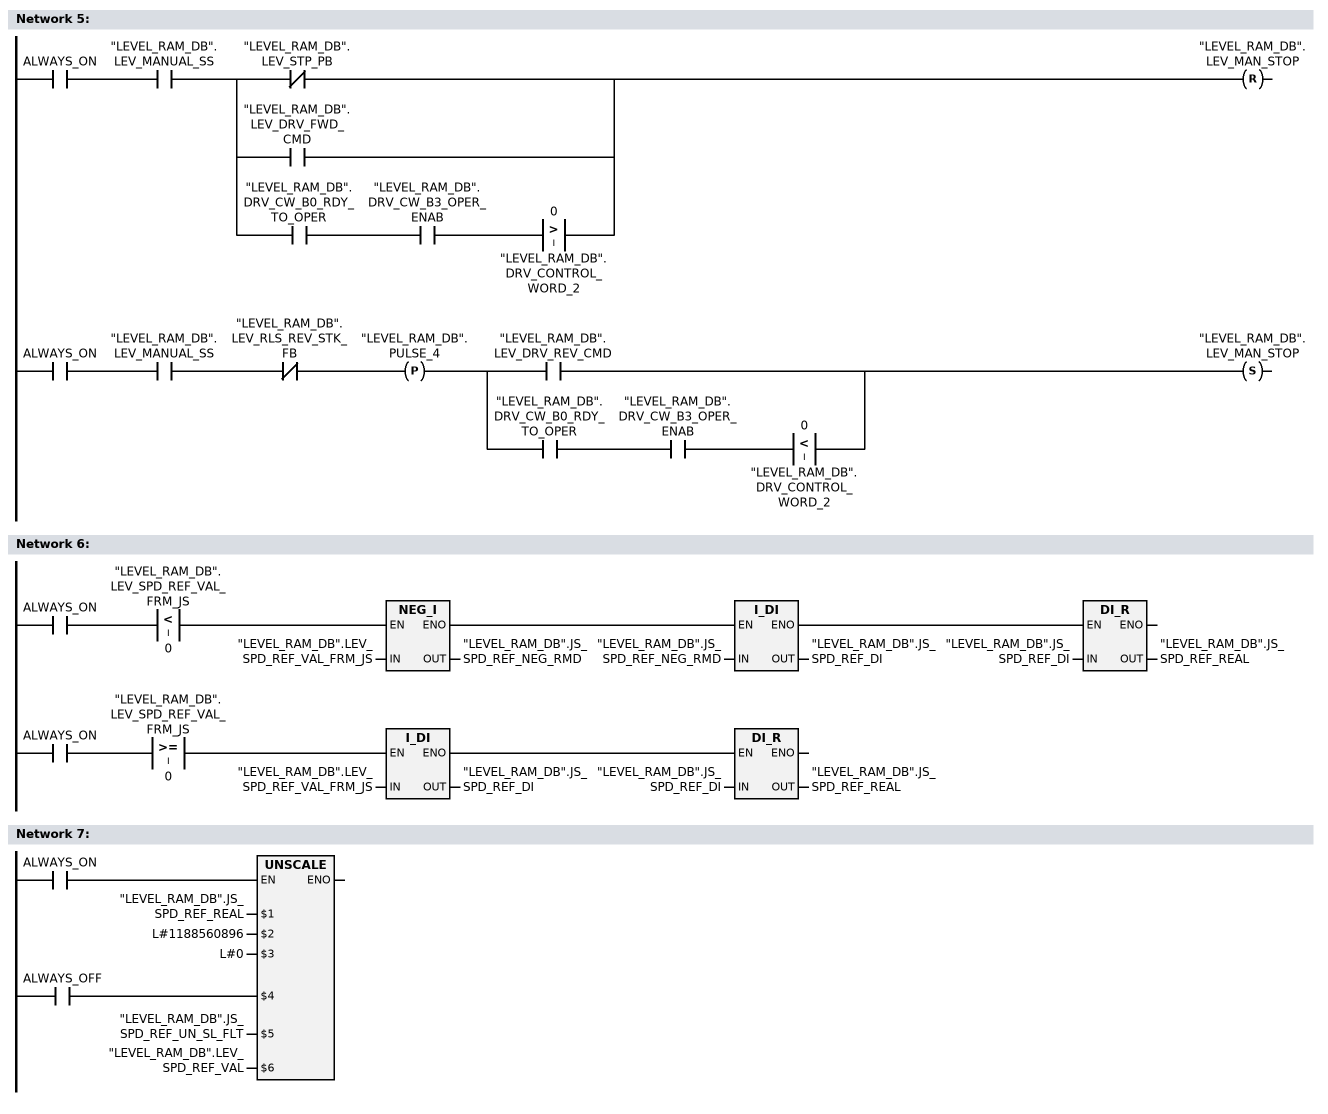
[picture p72: LEVELLER_RAM networks 5-7]
NETWORK
TITLE =
      A     "ALWAYS_ON";
      A     "LEVEL_RAM_DB".LEV_MANUAL_SS;
      =     L 0.0;
      A(;
      A     L 0.0;
      AN    "LEVEL_RAM_DB".LEV_RLS_REV_STK_FB;
      FP    "LEVEL_RAM_DB".PULSE_4;
      );
      A(;
      O     "LEVEL_RAM_DB".LEV_DRV_REV_CMD;
      O;
      A     "LEVEL_RAM_DB".DRV_CW_B0_RDY_TO_OPER;
      A     "LEVEL_RAM_DB".DRV_CW_B3_OPER_ENAB;
      A(;
      L     0;
      L     "LEVEL_RAM_DB".DRV_CONTROL_WORD_2;
      <I;
      );
      );
      S     "LEVEL_RAM_DB".LEV_MAN_STOP;
      A     L 0.0;
      A(;
      ON    "LEVEL_RAM_DB".LEV_STP_PB;
      O     "LEVEL_RAM_DB".LEV_DRV_FWD_CMD;
      O;
      A     "LEVEL_RAM_DB".DRV_CW_B0_RDY_TO_OPER;
      A     "LEVEL_RAM_DB".DRV_CW_B3_OPER_ENAB;
      A(;
      L     0;
      L     "LEVEL_RAM_DB".DRV_CONTROL_WORD_2;
      >I;
      );
      );
      R     "LEVEL_RAM_DB".LEV_MAN_STOP;
NETWORK
TITLE =
      A     "ALWAYS_ON";
      =     L 0.0;
      A(;
      A(;
      A     L 0.0;
      A(;
      L     "LEVEL_RAM_DB".LEV_SPD_REF_VAL_FRM_JS;
      L     0;
      <I;
      );
      JNB   M002;
      L     "LEVEL_RAM_DB".LEV_SPD_REF_VAL_FRM_JS;
      NEGI;
      T     "LEVEL_RAM_DB".JS_SPD_REF_NEG_RMD;
      AN    OV;
      SAVE;
      CLR;
M002: A     BR;
      );
      JNB   M003;
      L     "LEVEL_RAM_DB".JS_SPD_REF_NEG_RMD;
      ITD;
      T     "LEVEL_RAM_DB".JS_SPD_REF_DI;
      SET;
      SAVE;
      CLR;
M003: A     BR;
      );
      JNB   M004;
      L     "LEVEL_RAM_DB".JS_SPD_REF_DI;
      DTR;
      T     "LEVEL_RAM_DB".JS_SPD_REF_REAL;
M004: NOP   0;
      A(;
      A     L 0.0;
      A(;
      L     "LEVEL_RAM_DB".LEV_SPD_REF_VAL_FRM_JS;
      L     0;
      >=I;
      );
      JNB   M005;
      L     "LEVEL_RAM_DB".LEV_SPD_REF_VAL_FRM_JS;
      ITD;
      T     "LEVEL_RAM_DB".JS_SPD_REF_DI;
      SET;
      SAVE;
      CLR;
M005: A     BR;
      );
      JNB   M006;
      L     "LEVEL_RAM_DB".JS_SPD_REF_DI;
      DTR;
      T     "LEVEL_RAM_DB".JS_SPD_REF_REAL;
M006: NOP   0;
NETWORK
TITLE =
      A     "ALWAYS_OFF";
      =     L 0.0;
      BLD   103;
      A     "ALWAYS_ON";
      JNB   M007;
      CALL  "UNSCALE" (
           $1                       := "LEVEL_RAM_DB".JS_SPD_REF_REAL,
           $2                       := L#1188560896,
           $3                       := L#0,
           $4                       := L 0.0,
           $5                       := "LEVEL_RAM_DB".JS_SPD_REF_UN_SL_FLT,
           $6                       := "LEVEL_RAM_DB".LEV_SPD_REF_VAL);
M007: NOP   0;
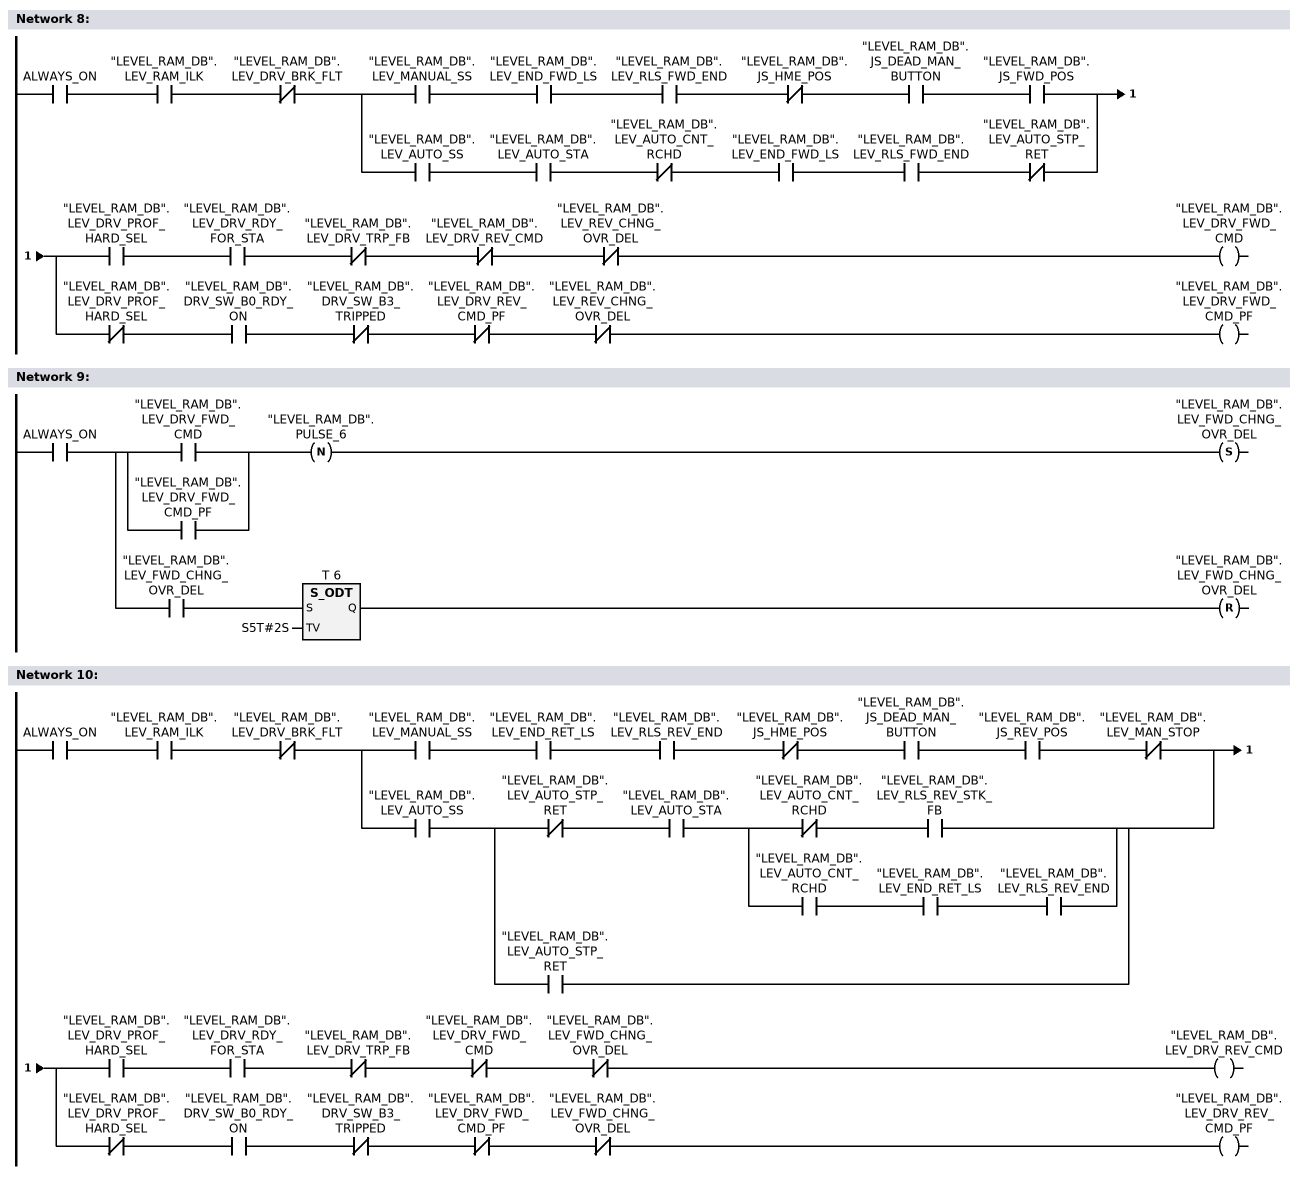
NETWORK
TITLE =
      A     "ALWAYS_ON";
      A     "LEVEL_RAM_DB".LEV_RAM_ILK;
      AN    "LEVEL_RAM_DB".LEV_DRV_BRK_FLT;
      A(;
      A     "LEVEL_RAM_DB".LEV_MANUAL_SS;
      A     "LEVEL_RAM_DB".LEV_END_FWD_LS;
      A     "LEVEL_RAM_DB".LEV_RLS_FWD_END;
      AN    "LEVEL_RAM_DB".JS_HME_POS;
      A     "LEVEL_RAM_DB".JS_DEAD_MAN_BUTTON;
      A     "LEVEL_RAM_DB".JS_FWD_POS;
      O;
      A     "LEVEL_RAM_DB".LEV_AUTO_SS;
      A     "LEVEL_RAM_DB".LEV_AUTO_STA;
      AN    "LEVEL_RAM_DB".LEV_AUTO_CNT_RCHD;
      A     "LEVEL_RAM_DB".LEV_END_FWD_LS;
      A     "LEVEL_RAM_DB".LEV_RLS_FWD_END;
      AN    "LEVEL_RAM_DB".LEV_AUTO_STP_RET;
      );
      =     L 0.0;
      A     L 0.0;
      A     "LEVEL_RAM_DB".LEV_DRV_PROF_HARD_SEL;
      A     "LEVEL_RAM_DB".LEV_DRV_RDY_FOR_STA;
      AN    "LEVEL_RAM_DB".LEV_DRV_TRP_FB;
      AN    "LEVEL_RAM_DB".LEV_DRV_REV_CMD;
      AN    "LEVEL_RAM_DB".LEV_REV_CHNG_OVR_DEL;
      =     "LEVEL_RAM_DB".LEV_DRV_FWD_CMD;
      A     L 0.0;
      AN    "LEVEL_RAM_DB".LEV_DRV_PROF_HARD_SEL;
      A     "LEVEL_RAM_DB".DRV_SW_B0_RDY_ON;
      AN    "LEVEL_RAM_DB".DRV_SW_B3_TRIPPED;
      AN    "LEVEL_RAM_DB".LEV_DRV_REV_CMD_PF;
      AN    "LEVEL_RAM_DB".LEV_REV_CHNG_OVR_DEL;
      =     "LEVEL_RAM_DB".LEV_DRV_FWD_CMD_PF;
NETWORK
TITLE =
      A     "ALWAYS_ON";
      =     L 0.0;
      A     L 0.0;
      A(;
      O     "LEVEL_RAM_DB".LEV_DRV_FWD_CMD;
      O     "LEVEL_RAM_DB".LEV_DRV_FWD_CMD_PF;
      );
      FN    "LEVEL_RAM_DB".PULSE_6;
      S     "LEVEL_RAM_DB".LEV_FWD_CHNG_OVR_DEL;
      A     L 0.0;
      A     "LEVEL_RAM_DB".LEV_FWD_CHNG_OVR_DEL;
      L     S5T#2S;
      SD    T 6;
      NOP   0;
      NOP   0;
      NOP   0;
      A     T 6;
      R     "LEVEL_RAM_DB".LEV_FWD_CHNG_OVR_DEL;
NETWORK
TITLE =
      A     "ALWAYS_ON";
      A     "LEVEL_RAM_DB".LEV_RAM_ILK;
      AN    "LEVEL_RAM_DB".LEV_DRV_BRK_FLT;
      A(;
      A     "LEVEL_RAM_DB".LEV_MANUAL_SS;
      A     "LEVEL_RAM_DB".LEV_END_RET_LS;
      A     "LEVEL_RAM_DB".LEV_RLS_REV_END;
      AN    "LEVEL_RAM_DB".JS_HME_POS;
      A     "LEVEL_RAM_DB".JS_DEAD_MAN_BUTTON;
      A     "LEVEL_RAM_DB".JS_REV_POS;
      AN    "LEVEL_RAM_DB".LEV_MAN_STOP;
      O;
      A     "LEVEL_RAM_DB".LEV_AUTO_SS;
      A(;
      AN    "LEVEL_RAM_DB".LEV_AUTO_STP_RET;
      A     "LEVEL_RAM_DB".LEV_AUTO_STA;
      A(;
      AN    "LEVEL_RAM_DB".LEV_AUTO_CNT_RCHD;
      A     "LEVEL_RAM_DB".LEV_RLS_REV_STK_FB;
      O;
      A     "LEVEL_RAM_DB".LEV_AUTO_CNT_RCHD;
      A     "LEVEL_RAM_DB".LEV_END_RET_LS;
      A     "LEVEL_RAM_DB".LEV_RLS_REV_END;
      );
      O     "LEVEL_RAM_DB".LEV_AUTO_STP_RET;
      );
      );
      =     L 0.0;
      A     L 0.0;
      A     "LEVEL_RAM_DB".LEV_DRV_PROF_HARD_SEL;
      A     "LEVEL_RAM_DB".LEV_DRV_RDY_FOR_STA;
      AN    "LEVEL_RAM_DB".LEV_DRV_TRP_FB;
      AN    "LEVEL_RAM_DB".LEV_DRV_FWD_CMD;
      AN    "LEVEL_RAM_DB".LEV_FWD_CHNG_OVR_DEL;
      =     "LEVEL_RAM_DB".LEV_DRV_REV_CMD;
      A     L 0.0;
      AN    "LEVEL_RAM_DB".LEV_DRV_PROF_HARD_SEL;
      A     "LEVEL_RAM_DB".DRV_SW_B0_RDY_ON;
      AN    "LEVEL_RAM_DB".DRV_SW_B3_TRIPPED;
      AN    "LEVEL_RAM_DB".LEV_DRV_FWD_CMD_PF;
      AN    "LEVEL_RAM_DB".LEV_FWD_CHNG_OVR_DEL;
      =     "LEVEL_RAM_DB".LEV_DRV_REV_CMD_PF;
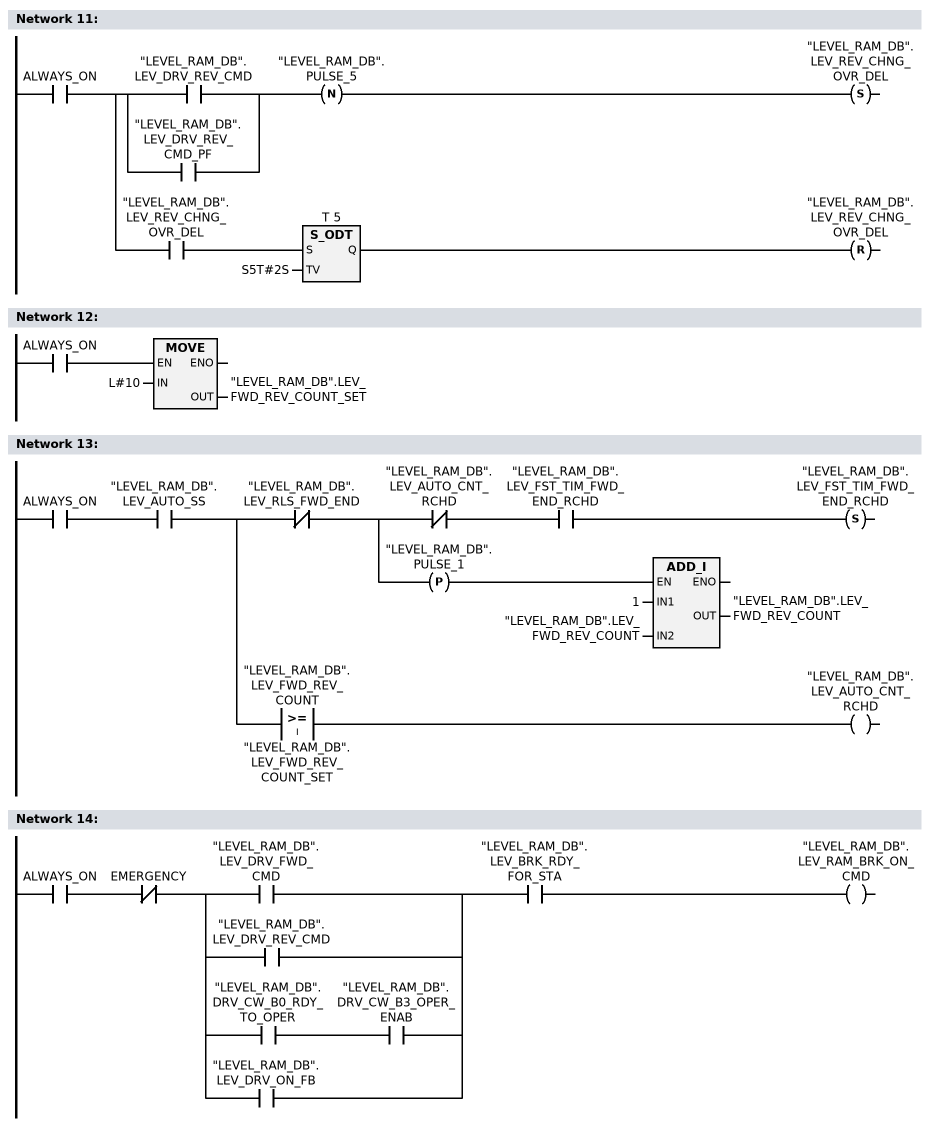
NETWORK
TITLE =
      A     "ALWAYS_ON";
      =     L 0.0;
      A     L 0.0;
      A(;
      O     "LEVEL_RAM_DB".LEV_DRV_REV_CMD;
      O     "LEVEL_RAM_DB".LEV_DRV_REV_CMD_PF;
      );
      FN    "LEVEL_RAM_DB".PULSE_5;
      S     "LEVEL_RAM_DB".LEV_REV_CHNG_OVR_DEL;
      A     L 0.0;
      A     "LEVEL_RAM_DB".LEV_REV_CHNG_OVR_DEL;
      L     S5T#2S;
      SD    T 5;
      NOP   0;
      NOP   0;
      NOP   0;
      A     T 5;
      R     "LEVEL_RAM_DB".LEV_REV_CHNG_OVR_DEL;
NETWORK
TITLE =
      A     "ALWAYS_ON";
      JNB   M008;
      L     L#10;
      T     "LEVEL_RAM_DB".LEV_FWD_REV_COUNT_SET;
M008: NOP   0;
NETWORK
TITLE =
      A     "ALWAYS_ON";
      A     "LEVEL_RAM_DB".LEV_AUTO_SS;
      =     L 0.0;
      A     L 0.0;
      AN    "LEVEL_RAM_DB".LEV_RLS_FWD_END;
      =     L 0.1;
      A     L 0.1;
      AN    "LEVEL_RAM_DB".LEV_AUTO_CNT_RCHD;
      A     "LEVEL_RAM_DB".LEV_FST_TIM_FWD_END_RCHD;
      S     "LEVEL_RAM_DB".LEV_FST_TIM_FWD_END_RCHD;
      A     L 0.1;
      FP    "LEVEL_RAM_DB".PULSE_1;
      JNB   M009;
      L     1;
      L     "LEVEL_RAM_DB".LEV_FWD_REV_COUNT;
      +I;
      T     "LEVEL_RAM_DB".LEV_FWD_REV_COUNT;
M009: NOP   0;
      A     L 0.0;
      A(;
      L     "LEVEL_RAM_DB".LEV_FWD_REV_COUNT;
      L     "LEVEL_RAM_DB".LEV_FWD_REV_COUNT_SET;
      >=I;
      );
      =     "LEVEL_RAM_DB".LEV_AUTO_CNT_RCHD;
NETWORK
TITLE =
      A     "ALWAYS_ON";
      AN    "EMERGENCY";
      A(;
      O     "LEVEL_RAM_DB".LEV_DRV_FWD_CMD;
      O     "LEVEL_RAM_DB".LEV_DRV_REV_CMD;
      O;
      A     "LEVEL_RAM_DB".DRV_CW_B0_RDY_TO_OPER;
      A     "LEVEL_RAM_DB".DRV_CW_B3_OPER_ENAB;
      O     "LEVEL_RAM_DB".LEV_DRV_ON_FB;
      );
      A     "LEVEL_RAM_DB".LEV_BRK_RDY_FOR_STA;
      =     "LEVEL_RAM_DB".LEV_RAM_BRK_ON_CMD;
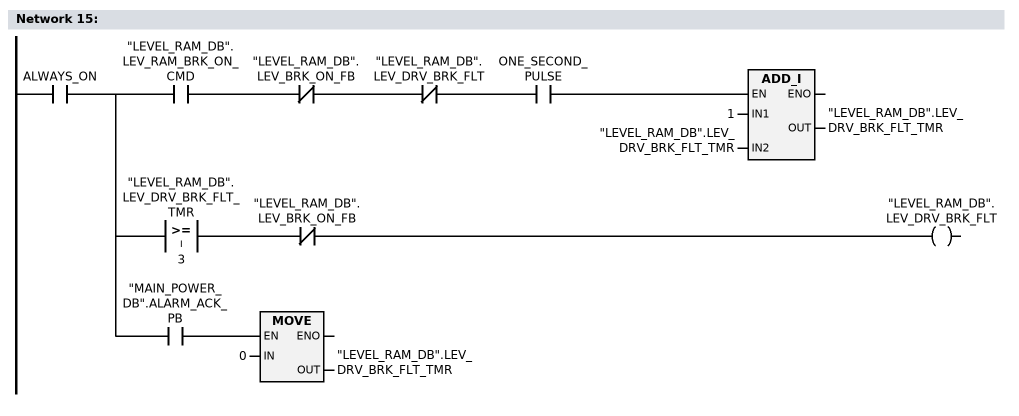
NETWORK
TITLE =
      A     "ALWAYS_ON";
      =     L 0.0;
      A     L 0.0;
      A     "LEVEL_RAM_DB".LEV_RAM_BRK_ON_CMD;
      AN    "LEVEL_RAM_DB".LEV_BRK_ON_FB;
      AN    "LEVEL_RAM_DB".LEV_DRV_BRK_FLT;
      A     "ONE_SECOND_PULSE";
      JNB   M010;
      L     1;
      L     "LEVEL_RAM_DB".LEV_DRV_BRK_FLT_TMR;
      +I;
      T     "LEVEL_RAM_DB".LEV_DRV_BRK_FLT_TMR;
M010: NOP   0;
      A     L 0.0;
      A(;
      L     "LEVEL_RAM_DB".LEV_DRV_BRK_FLT_TMR;
      L     3;
      >=I;
      );
      AN    "LEVEL_RAM_DB".LEV_BRK_ON_FB;
      =     "LEVEL_RAM_DB".LEV_DRV_BRK_FLT;
      A     L 0.0;
      A     "MAIN_POWER_DB".ALARM_ACK_PB;
      JNB   M011;
      L     0;
      T     "LEVEL_RAM_DB".LEV_DRV_BRK_FLT_TMR;
M011: NOP   0;
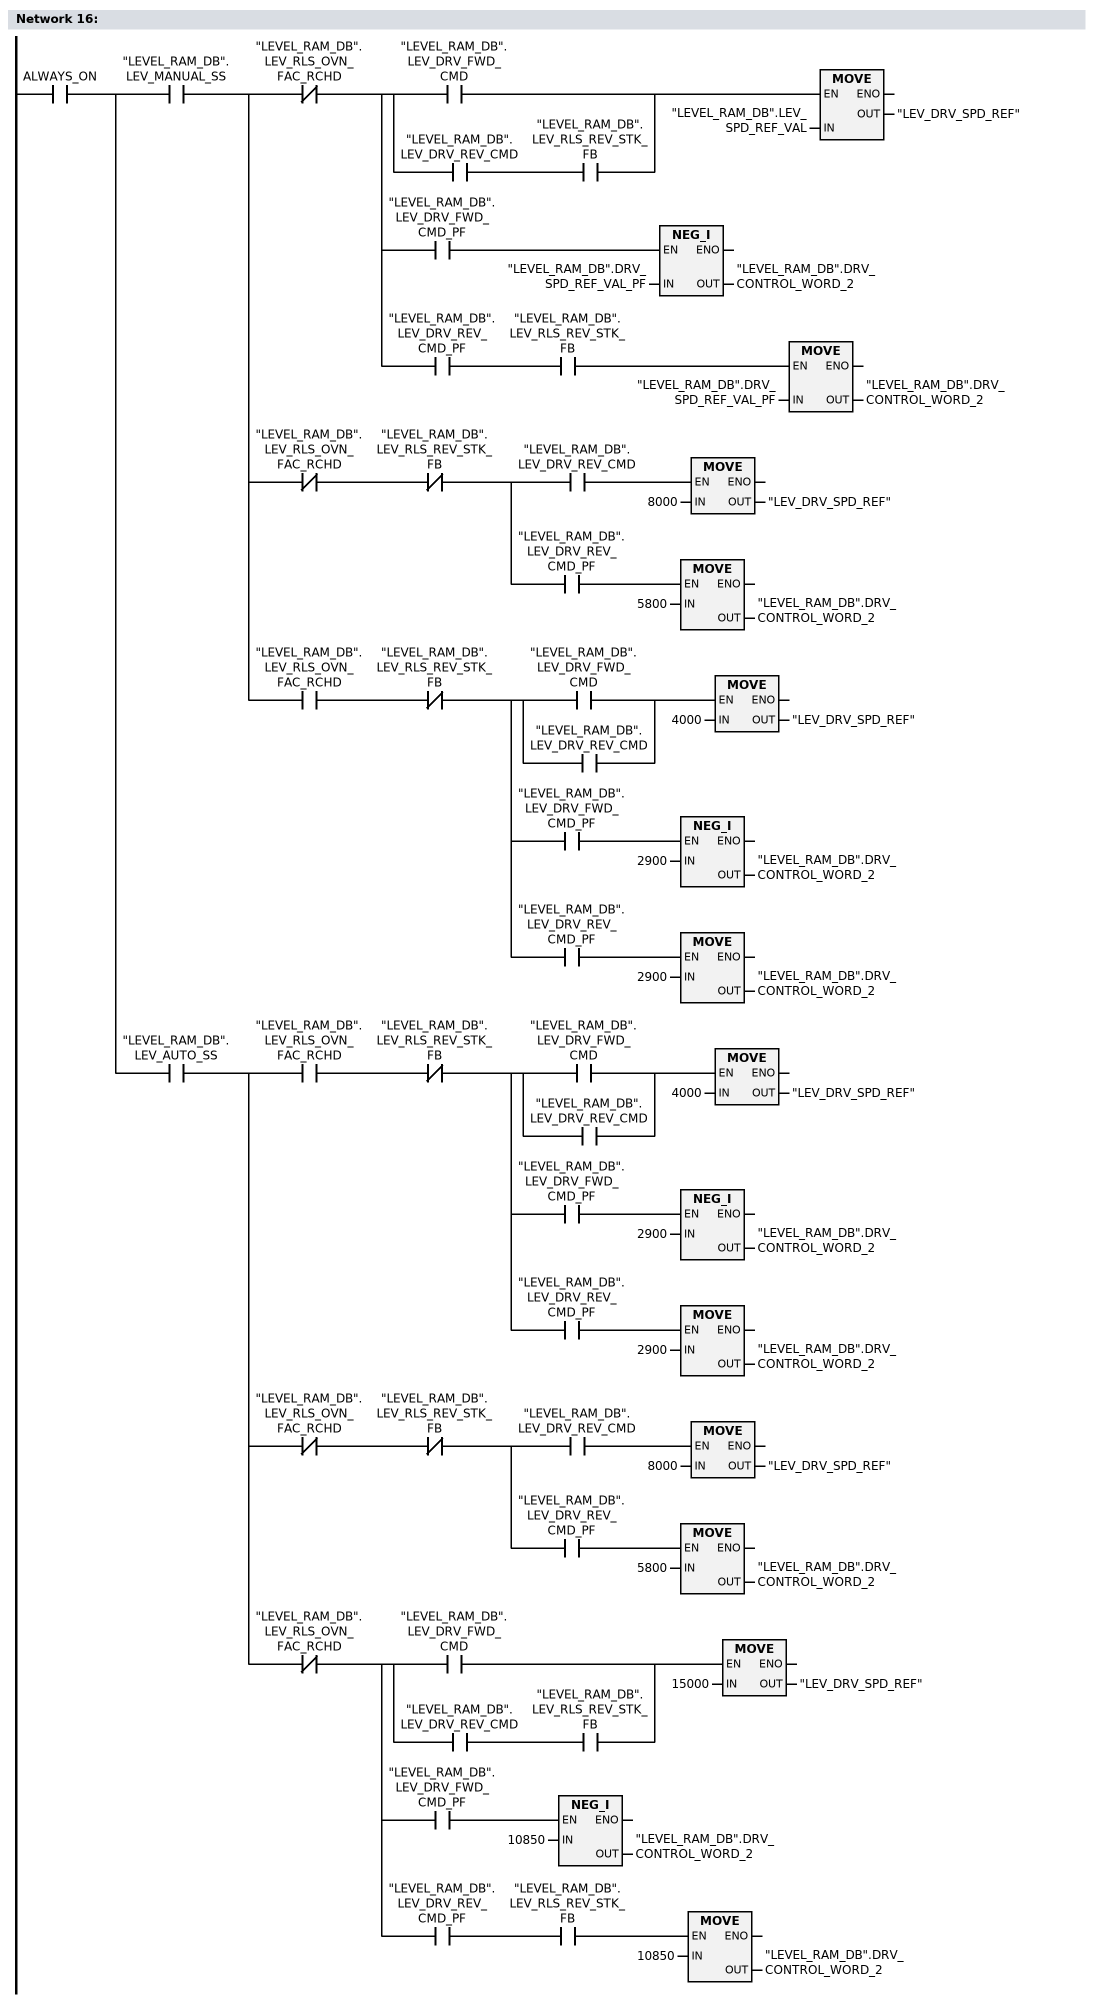
NETWORK
TITLE =
      A     "ALWAYS_ON";
      =     L 0.0;
      A     L 0.0;
      A     "LEVEL_RAM_DB".LEV_MANUAL_SS;
      =     L 0.1;
      A     L 0.1;
      AN    "LEVEL_RAM_DB".LEV_RLS_OVN_FAC_RCHD;
      =     L 0.2;
      A     L 0.2;
      A(;
      O     "LEVEL_RAM_DB".LEV_DRV_FWD_CMD;
      O;
      A     "LEVEL_RAM_DB".LEV_DRV_REV_CMD;
      A     "LEVEL_RAM_DB".LEV_RLS_REV_STK_FB;
      );
      JNB   M012;
      L     "LEVEL_RAM_DB".LEV_SPD_REF_VAL;
      T     "LEV_DRV_SPD_REF";
M012: NOP   0;
      A     L 0.2;
      A     "LEVEL_RAM_DB".LEV_DRV_FWD_CMD_PF;
      JNB   M013;
      L     "LEVEL_RAM_DB".DRV_SPD_REF_VAL_PF;
      NEGI;
      T     "LEVEL_RAM_DB".DRV_CONTROL_WORD_2;
M013: NOP   0;
      A     L 0.2;
      A     "LEVEL_RAM_DB".LEV_DRV_REV_CMD_PF;
      A     "LEVEL_RAM_DB".LEV_RLS_REV_STK_FB;
      JNB   M014;
      L     "LEVEL_RAM_DB".DRV_SPD_REF_VAL_PF;
      T     "LEVEL_RAM_DB".DRV_CONTROL_WORD_2;
M014: NOP   0;
      A     L 0.1;
      AN    "LEVEL_RAM_DB".LEV_RLS_OVN_FAC_RCHD;
      AN    "LEVEL_RAM_DB".LEV_RLS_REV_STK_FB;
      =     L 0.2;
      A     L 0.2;
      A     "LEVEL_RAM_DB".LEV_DRV_REV_CMD;
      JNB   M015;
      L     8000;
      T     "LEV_DRV_SPD_REF";
M015: NOP   0;
      A     L 0.2;
      A     "LEVEL_RAM_DB".LEV_DRV_REV_CMD_PF;
      JNB   M016;
      L     5800;
      T     "LEVEL_RAM_DB".DRV_CONTROL_WORD_2;
M016: NOP   0;
      A     L 0.1;
      A     "LEVEL_RAM_DB".LEV_RLS_OVN_FAC_RCHD;
      AN    "LEVEL_RAM_DB".LEV_RLS_REV_STK_FB;
      =     L 0.2;
      A     L 0.2;
      A(;
      O     "LEVEL_RAM_DB".LEV_DRV_FWD_CMD;
      O     "LEVEL_RAM_DB".LEV_DRV_REV_CMD;
      );
      JNB   M017;
      L     4000;
      T     "LEV_DRV_SPD_REF";
M017: NOP   0;
      A     L 0.2;
      A     "LEVEL_RAM_DB".LEV_DRV_FWD_CMD_PF;
      JNB   M018;
      L     2900;
      NEGI;
      T     "LEVEL_RAM_DB".DRV_CONTROL_WORD_2;
M018: NOP   0;
      A     L 0.2;
      A     "LEVEL_RAM_DB".LEV_DRV_REV_CMD_PF;
      JNB   M019;
      L     2900;
      T     "LEVEL_RAM_DB".DRV_CONTROL_WORD_2;
M019: NOP   0;
      A     L 0.0;
      A     "LEVEL_RAM_DB".LEV_AUTO_SS;
      =     L 0.1;
      A     L 0.1;
      A     "LEVEL_RAM_DB".LEV_RLS_OVN_FAC_RCHD;
      AN    "LEVEL_RAM_DB".LEV_RLS_REV_STK_FB;
      =     L 0.2;
      A     L 0.2;
      A(;
      O     "LEVEL_RAM_DB".LEV_DRV_FWD_CMD;
      O     "LEVEL_RAM_DB".LEV_DRV_REV_CMD;
      );
      JNB   M020;
      L     4000;
      T     "LEV_DRV_SPD_REF";
M020: NOP   0;
      A     L 0.2;
      A     "LEVEL_RAM_DB".LEV_DRV_FWD_CMD_PF;
      JNB   M021;
      L     2900;
      NEGI;
      T     "LEVEL_RAM_DB".DRV_CONTROL_WORD_2;
M021: NOP   0;
      A     L 0.2;
      A     "LEVEL_RAM_DB".LEV_DRV_REV_CMD_PF;
      JNB   M022;
      L     2900;
      T     "LEVEL_RAM_DB".DRV_CONTROL_WORD_2;
M022: NOP   0;
      A     L 0.1;
      AN    "LEVEL_RAM_DB".LEV_RLS_OVN_FAC_RCHD;
      AN    "LEVEL_RAM_DB".LEV_RLS_REV_STK_FB;
      =     L 0.2;
      A     L 0.2;
      A     "LEVEL_RAM_DB".LEV_DRV_REV_CMD;
      JNB   M023;
      L     8000;
      T     "LEV_DRV_SPD_REF";
M023: NOP   0;
      A     L 0.2;
      A     "LEVEL_RAM_DB".LEV_DRV_REV_CMD_PF;
      JNB   M024;
      L     5800;
      T     "LEVEL_RAM_DB".DRV_CONTROL_WORD_2;
M024: NOP   0;
      A     L 0.1;
      AN    "LEVEL_RAM_DB".LEV_RLS_OVN_FAC_RCHD;
      =     L 0.2;
      A     L 0.2;
      A(;
      O     "LEVEL_RAM_DB".LEV_DRV_FWD_CMD;
      O;
      A     "LEVEL_RAM_DB".LEV_DRV_REV_CMD;
      A     "LEVEL_RAM_DB".LEV_RLS_REV_STK_FB;
      );
      JNB   M025;
      L     15000;
      T     "LEV_DRV_SPD_REF";
M025: NOP   0;
      A     L 0.2;
      A     "LEVEL_RAM_DB".LEV_DRV_FWD_CMD_PF;
      JNB   M026;
      L     10850;
      NEGI;
      T     "LEVEL_RAM_DB".DRV_CONTROL_WORD_2;
M026: NOP   0;
      A     L 0.2;
      A     "LEVEL_RAM_DB".LEV_DRV_REV_CMD_PF;
      A     "LEVEL_RAM_DB".LEV_RLS_REV_STK_FB;
      JNB   M027;
      L     10850;
      T     "LEVEL_RAM_DB".DRV_CONTROL_WORD_2;
M027: NOP   0;
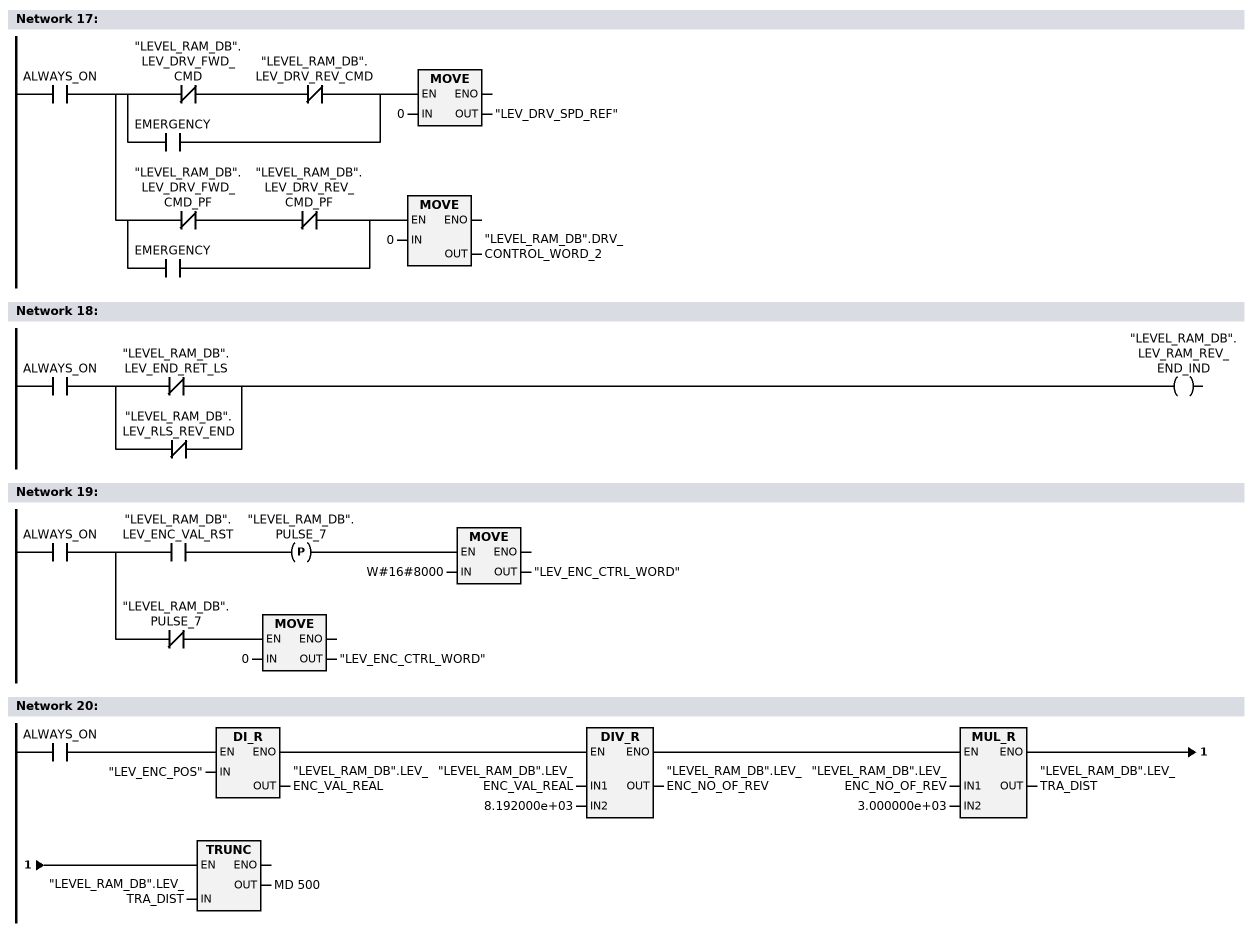
NETWORK
TITLE =
      A     "ALWAYS_ON";
      =     L 0.0;
      A     L 0.0;
      A(;
      AN    "LEVEL_RAM_DB".LEV_DRV_FWD_CMD;
      AN    "LEVEL_RAM_DB".LEV_DRV_REV_CMD;
      O     "EMERGENCY";
      );
      JNB   M028;
      L     0;
      T     "LEV_DRV_SPD_REF";
M028: NOP   0;
      A     L 0.0;
      A(;
      AN    "LEVEL_RAM_DB".LEV_DRV_FWD_CMD_PF;
      AN    "LEVEL_RAM_DB".LEV_DRV_REV_CMD_PF;
      O     "EMERGENCY";
      );
      JNB   M029;
      L     0;
      T     "LEVEL_RAM_DB".DRV_CONTROL_WORD_2;
M029: NOP   0;
NETWORK
TITLE =
      A     "ALWAYS_ON";
      A(;
      ON    "LEVEL_RAM_DB".LEV_END_RET_LS;
      ON    "LEVEL_RAM_DB".LEV_RLS_REV_END;
      );
      =     "LEVEL_RAM_DB".LEV_RAM_REV_END_IND;
NETWORK
TITLE =
      A     "ALWAYS_ON";
      =     L 0.0;
      A     L 0.0;
      A     "LEVEL_RAM_DB".LEV_ENC_VAL_RST;
      FP    "LEVEL_RAM_DB".PULSE_7;
      JNB   M030;
      L     W#16#8000;
      T     "LEV_ENC_CTRL_WORD";
M030: NOP   0;
      A     L 0.0;
      AN    "LEVEL_RAM_DB".PULSE_7;
      JNB   M031;
      L     0;
      T     "LEV_ENC_CTRL_WORD";
M031: NOP   0;
NETWORK
TITLE =
      A(;
      A(;
      A(;
      A     "ALWAYS_ON";
      JNB   M032;
      L     "LEV_ENC_POS";
      DTR;
      T     "LEVEL_RAM_DB".LEV_ENC_VAL_REAL;
      SET;
      SAVE;
      CLR;
M032: A     BR;
      );
      JNB   M033;
      L     "LEVEL_RAM_DB".LEV_ENC_VAL_REAL;
      L     8.192000e+03;
      /R;
      T     "LEVEL_RAM_DB".LEV_ENC_NO_OF_REV;
      AN    OV;
      SAVE;
      CLR;
M033: A     BR;
      );
      JNB   M034;
      L     "LEVEL_RAM_DB".LEV_ENC_NO_OF_REV;
      L     3.000000e+03;
      *R;
      T     "LEVEL_RAM_DB".LEV_TRA_DIST;
      AN    OV;
      SAVE;
      CLR;
M034: A     BR;
      );
      JNB   M035;
      L     "LEVEL_RAM_DB".LEV_TRA_DIST;
      TRUNC;
      T     MD 500;
M035: NOP   0;
END_FUNCTION

FUNCTION "LEVELER_DOOR" : VOID	// FC 6
AUTHOR : Kamillas
VERSION : 0.1
BEGIN
// (block stored without names or comments; labels and parameter names are numbered)
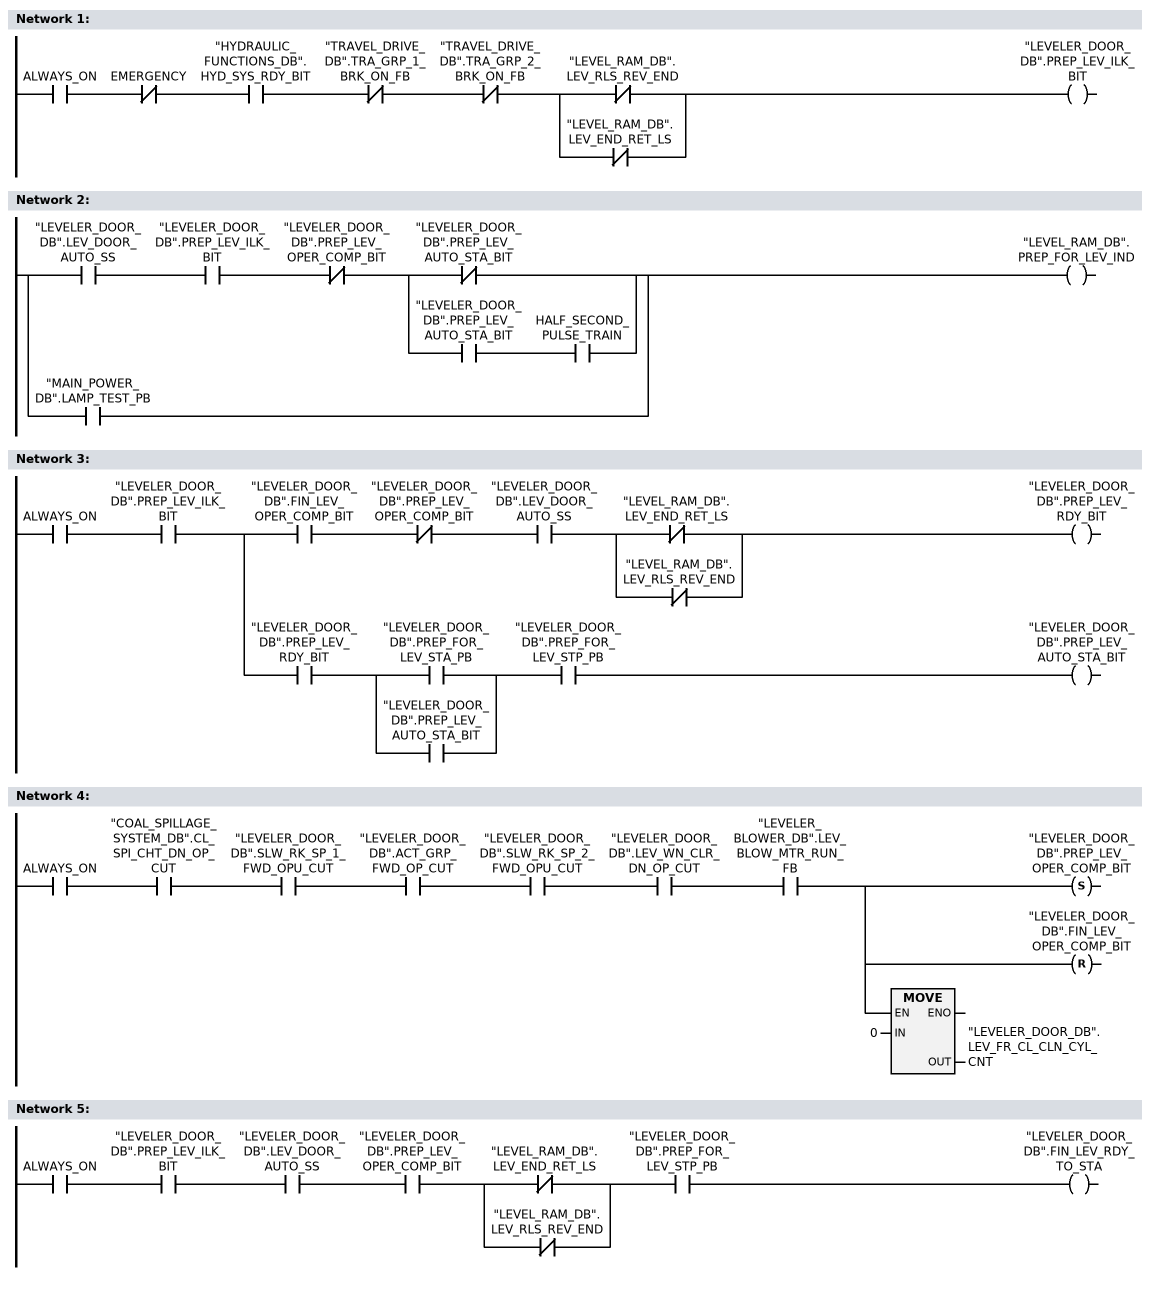
NETWORK
TITLE =
      A     "ALWAYS_ON";
      AN    "EMERGENCY";
      A     "HYDRAULIC_FUNCTIONS_DB".HYD_SYS_RDY_BIT;
      AN    "TRAVEL_DRIVE_DB".TRA_GRP_1_BRK_ON_FB;
      AN    "TRAVEL_DRIVE_DB".TRA_GRP_2_BRK_ON_FB;
      A(;
      ON    "LEVEL_RAM_DB".LEV_RLS_REV_END;
      ON    "LEVEL_RAM_DB".LEV_END_RET_LS;
      );
      =     "LEVELER_DOOR_DB".PREP_LEV_ILK_BIT;
NETWORK
TITLE =
      A     "LEVELER_DOOR_DB".LEV_DOOR_AUTO_SS;
      A     "LEVELER_DOOR_DB".PREP_LEV_ILK_BIT;
      AN    "LEVELER_DOOR_DB".PREP_LEV_OPER_COMP_BIT;
      A(;
      ON    "LEVELER_DOOR_DB".PREP_LEV_AUTO_STA_BIT;
      O;
      A     "LEVELER_DOOR_DB".PREP_LEV_AUTO_STA_BIT;
      A     "HALF_SECOND_PULSE_TRAIN";
      );
      O     "MAIN_POWER_DB".LAMP_TEST_PB;
      =     "LEVEL_RAM_DB".PREP_FOR_LEV_IND;
NETWORK
TITLE =
      A     "ALWAYS_ON";
      A     "LEVELER_DOOR_DB".PREP_LEV_ILK_BIT;
      =     L 0.0;
      A     L 0.0;
      A     "LEVELER_DOOR_DB".FIN_LEV_OPER_COMP_BIT;
      AN    "LEVELER_DOOR_DB".PREP_LEV_OPER_COMP_BIT;
      A     "LEVELER_DOOR_DB".LEV_DOOR_AUTO_SS;
      A(;
      ON    "LEVEL_RAM_DB".LEV_END_RET_LS;
      ON    "LEVEL_RAM_DB".LEV_RLS_REV_END;
      );
      =     "LEVELER_DOOR_DB".PREP_LEV_RDY_BIT;
      A     L 0.0;
      A     "LEVELER_DOOR_DB".PREP_LEV_RDY_BIT;
      A(;
      O     "LEVELER_DOOR_DB".PREP_FOR_LEV_STA_PB;
      O     "LEVELER_DOOR_DB".PREP_LEV_AUTO_STA_BIT;
      );
      A     "LEVELER_DOOR_DB".PREP_FOR_LEV_STP_PB;
      =     "LEVELER_DOOR_DB".PREP_LEV_AUTO_STA_BIT;
NETWORK
TITLE =
      A     "ALWAYS_ON";
      A     "COAL_SPILLAGE_SYSTEM_DB".CL_SPI_CHT_DN_OP_CUT;
      A     "LEVELER_DOOR_DB".SLW_RK_SP_1_FWD_OPU_CUT;
      A     "LEVELER_DOOR_DB".ACT_GRP_FWD_OP_CUT;
      A     "LEVELER_DOOR_DB".SLW_RK_SP_2_FWD_OPU_CUT;
      A     "LEVELER_DOOR_DB".LEV_WN_CLR_DN_OP_CUT;
      A     "LEVELER_BLOWER_DB".LEV_BLOW_MTR_RUN_FB;
      =     L 0.0;
      A     L 0.0;
      BLD   102;
      S     "LEVELER_DOOR_DB".PREP_LEV_OPER_COMP_BIT;
      A     L 0.0;
      BLD   102;
      R     "LEVELER_DOOR_DB".FIN_LEV_OPER_COMP_BIT;
      A     L 0.0;
      JNB   M001;
      L     0;
      T     "LEVELER_DOOR_DB".LEV_FR_CL_CLN_CYL_CNT;
M001: NOP   0;
NETWORK
TITLE =
      A     "ALWAYS_ON";
      A     "LEVELER_DOOR_DB".PREP_LEV_ILK_BIT;
      A     "LEVELER_DOOR_DB".LEV_DOOR_AUTO_SS;
      A     "LEVELER_DOOR_DB".PREP_LEV_OPER_COMP_BIT;
      A(;
      ON    "LEVEL_RAM_DB".LEV_END_RET_LS;
      ON    "LEVEL_RAM_DB".LEV_RLS_REV_END;
      );
      A     "LEVELER_DOOR_DB".PREP_FOR_LEV_STP_PB;
      =     "LEVELER_DOOR_DB".FIN_LEV_RDY_TO_STA;
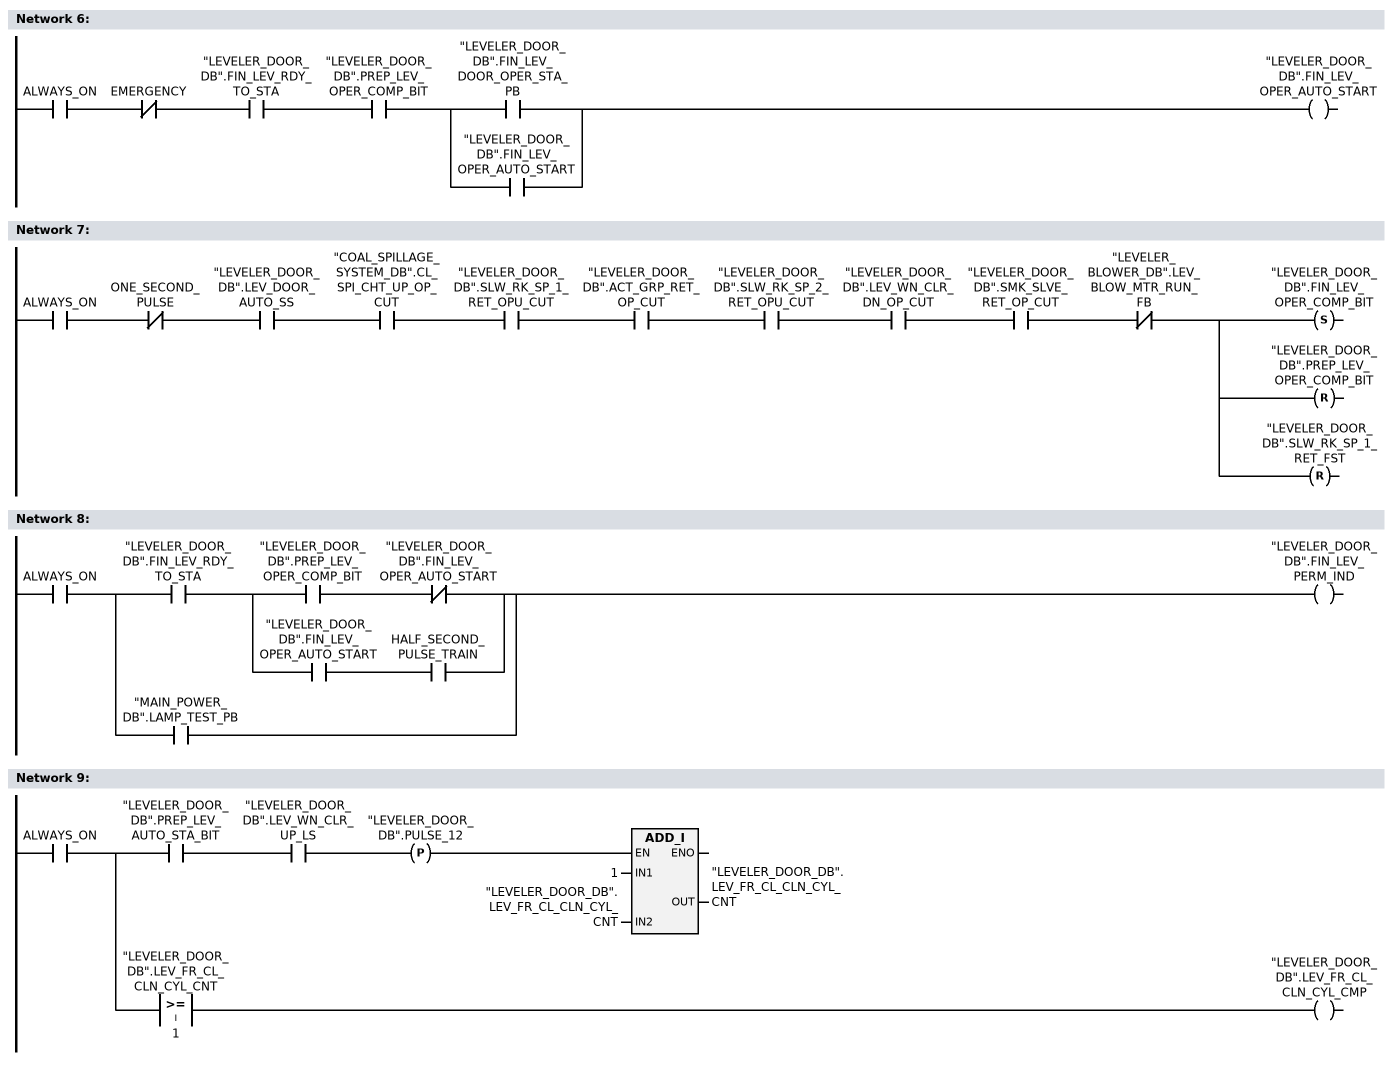
NETWORK
TITLE =
      A     "ALWAYS_ON";
      AN    "EMERGENCY";
      A     "LEVELER_DOOR_DB".FIN_LEV_RDY_TO_STA;
      A     "LEVELER_DOOR_DB".PREP_LEV_OPER_COMP_BIT;
      A(;
      O     "LEVELER_DOOR_DB".FIN_LEV_DOOR_OPER_STA_PB;
      O     "LEVELER_DOOR_DB".FIN_LEV_OPER_AUTO_START;
      );
      =     "LEVELER_DOOR_DB".FIN_LEV_OPER_AUTO_START;
NETWORK
TITLE =
      A     "ALWAYS_ON";
      AN    "ONE_SECOND_PULSE";
      A     "LEVELER_DOOR_DB".LEV_DOOR_AUTO_SS;
      A     "COAL_SPILLAGE_SYSTEM_DB".CL_SPI_CHT_UP_OP_CUT;
      A     "LEVELER_DOOR_DB".SLW_RK_SP_1_RET_OPU_CUT;
      A     "LEVELER_DOOR_DB".ACT_GRP_RET_OP_CUT;
      A     "LEVELER_DOOR_DB".SLW_RK_SP_2_RET_OPU_CUT;
      A     "LEVELER_DOOR_DB".LEV_WN_CLR_DN_OP_CUT;
      A     "LEVELER_DOOR_DB".SMK_SLVE_RET_OP_CUT;
      AN    "LEVELER_BLOWER_DB".LEV_BLOW_MTR_RUN_FB;
      S     "LEVELER_DOOR_DB".FIN_LEV_OPER_COMP_BIT;
      R     "LEVELER_DOOR_DB".PREP_LEV_OPER_COMP_BIT;
      R     "LEVELER_DOOR_DB".SLW_RK_SP_1_RET_FST;
NETWORK
TITLE =
      A     "ALWAYS_ON";
      A(;
      A     "LEVELER_DOOR_DB".FIN_LEV_RDY_TO_STA;
      A(;
      A     "LEVELER_DOOR_DB".PREP_LEV_OPER_COMP_BIT;
      AN    "LEVELER_DOOR_DB".FIN_LEV_OPER_AUTO_START;
      O;
      A     "LEVELER_DOOR_DB".FIN_LEV_OPER_AUTO_START;
      A     "HALF_SECOND_PULSE_TRAIN";
      );
      O     "MAIN_POWER_DB".LAMP_TEST_PB;
      );
      =     "LEVELER_DOOR_DB".FIN_LEV_PERM_IND;
NETWORK
TITLE =
      A     "ALWAYS_ON";
      =     L 0.0;
      A     L 0.0;
      A     "LEVELER_DOOR_DB".PREP_LEV_AUTO_STA_BIT;
      A     "LEVELER_DOOR_DB".LEV_WN_CLR_UP_LS;
      FP    "LEVELER_DOOR_DB".PULSE_12;
      JNB   M002;
      L     1;
      L     "LEVELER_DOOR_DB".LEV_FR_CL_CLN_CYL_CNT;
      +I;
      T     "LEVELER_DOOR_DB".LEV_FR_CL_CLN_CYL_CNT;
M002: NOP   0;
      A     L 0.0;
      A(;
      L     "LEVELER_DOOR_DB".LEV_FR_CL_CLN_CYL_CNT;
      L     1;
      >=I;
      );
      =     "LEVELER_DOOR_DB".LEV_FR_CL_CLN_CYL_CMP;
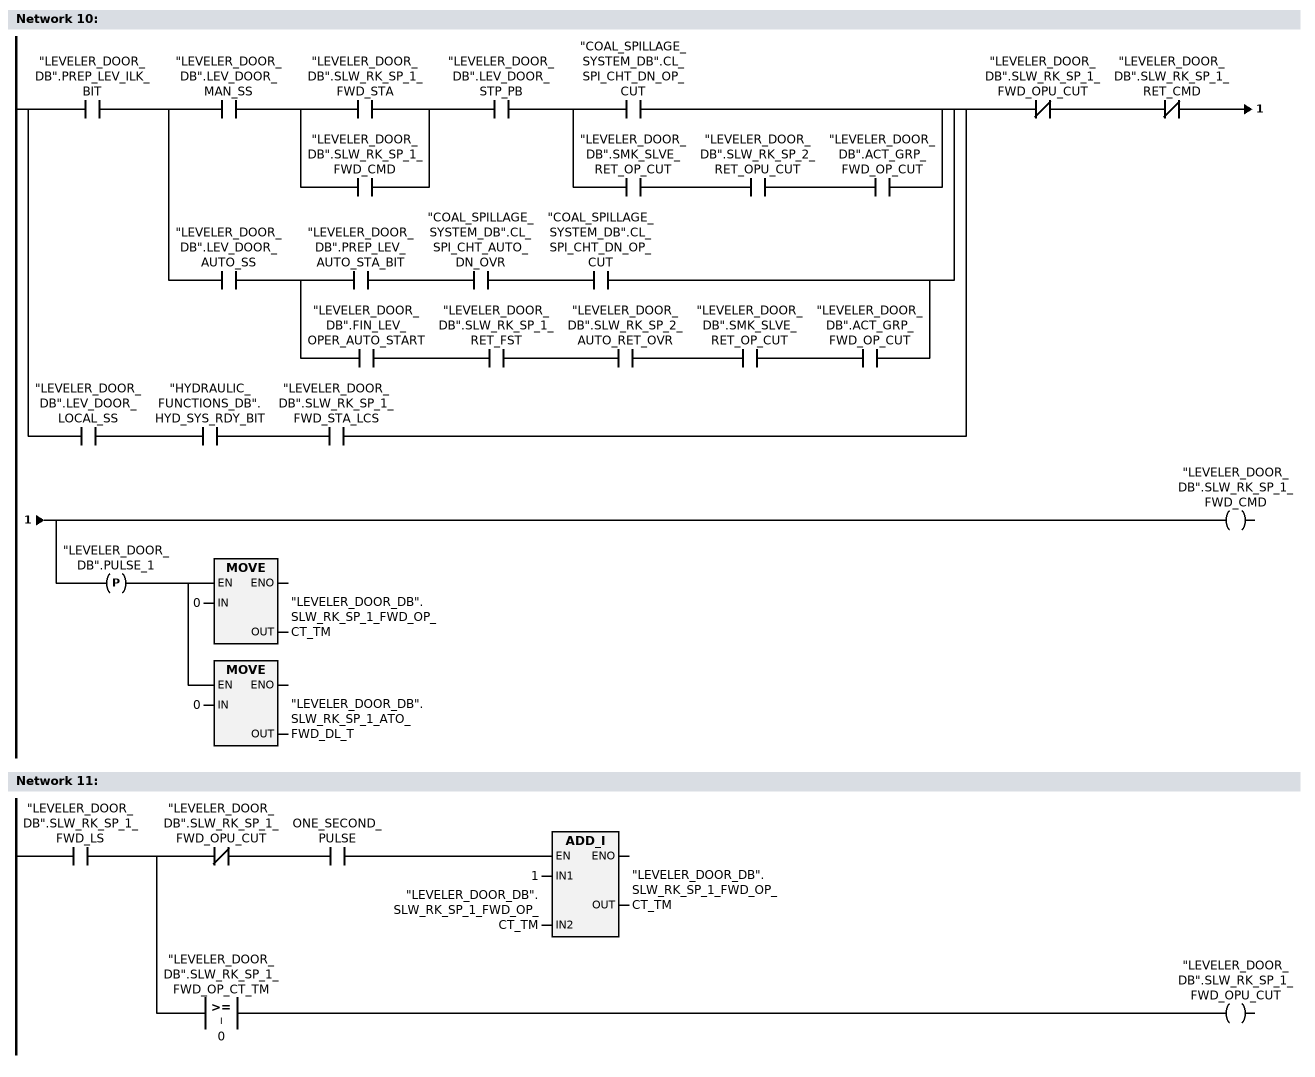
NETWORK
TITLE =
      A(;
      A     "LEVELER_DOOR_DB".PREP_LEV_ILK_BIT;
      A(;
      A     "LEVELER_DOOR_DB".LEV_DOOR_MAN_SS;
      A(;
      O     "LEVELER_DOOR_DB".SLW_RK_SP_1_FWD_STA;
      O     "LEVELER_DOOR_DB".SLW_RK_SP_1_FWD_CMD;
      );
      A     "LEVELER_DOOR_DB".LEV_DOOR_STP_PB;
      A(;
      O     "COAL_SPILLAGE_SYSTEM_DB".CL_SPI_CHT_DN_OP_CUT;
      O;
      A     "LEVELER_DOOR_DB".SMK_SLVE_RET_OP_CUT;
      A     "LEVELER_DOOR_DB".SLW_RK_SP_2_RET_OPU_CUT;
      A     "LEVELER_DOOR_DB".ACT_GRP_FWD_OP_CUT;
      );
      O;
      A     "LEVELER_DOOR_DB".LEV_DOOR_AUTO_SS;
      A(;
      A     "LEVELER_DOOR_DB".PREP_LEV_AUTO_STA_BIT;
      A     "COAL_SPILLAGE_SYSTEM_DB".CL_SPI_CHT_AUTO_DN_OVR;
      A     "COAL_SPILLAGE_SYSTEM_DB".CL_SPI_CHT_DN_OP_CUT;
      O;
      A     "LEVELER_DOOR_DB".FIN_LEV_OPER_AUTO_START;
      A     "LEVELER_DOOR_DB".SLW_RK_SP_1_RET_FST;
      A     "LEVELER_DOOR_DB".SLW_RK_SP_2_AUTO_RET_OVR;
      A     "LEVELER_DOOR_DB".SMK_SLVE_RET_OP_CUT;
      A     "LEVELER_DOOR_DB".ACT_GRP_FWD_OP_CUT;
      );
      );
      O;
      A     "LEVELER_DOOR_DB".LEV_DOOR_LOCAL_SS;
      A     "HYDRAULIC_FUNCTIONS_DB".HYD_SYS_RDY_BIT;
      A     "LEVELER_DOOR_DB".SLW_RK_SP_1_FWD_STA_LCS;
      );
      AN    "LEVELER_DOOR_DB".SLW_RK_SP_1_FWD_OPU_CUT;
      AN    "LEVELER_DOOR_DB".SLW_RK_SP_1_RET_CMD;
      =     L 0.0;
      A     L 0.0;
      BLD   102;
      =     "LEVELER_DOOR_DB".SLW_RK_SP_1_FWD_CMD;
      A     L 0.0;
      FP    "LEVELER_DOOR_DB".PULSE_1;
      =     L 0.1;
      A     L 0.1;
      JNB   M003;
      L     0;
      T     "LEVELER_DOOR_DB".SLW_RK_SP_1_FWD_OP_CT_TM;
M003: NOP   0;
      A     L 0.1;
      JNB   M004;
      L     0;
      T     "LEVELER_DOOR_DB".SLW_RK_SP_1_ATO_FWD_DL_T;
M004: NOP   0;
NETWORK
TITLE =
      A     "LEVELER_DOOR_DB".SLW_RK_SP_1_FWD_LS;
      =     L 0.0;
      A     L 0.0;
      AN    "LEVELER_DOOR_DB".SLW_RK_SP_1_FWD_OPU_CUT;
      A     "ONE_SECOND_PULSE";
      JNB   M005;
      L     1;
      L     "LEVELER_DOOR_DB".SLW_RK_SP_1_FWD_OP_CT_TM;
      +I;
      T     "LEVELER_DOOR_DB".SLW_RK_SP_1_FWD_OP_CT_TM;
M005: NOP   0;
      A     L 0.0;
      A(;
      L     "LEVELER_DOOR_DB".SLW_RK_SP_1_FWD_OP_CT_TM;
      L     0;
      >=I;
      );
      =     "LEVELER_DOOR_DB".SLW_RK_SP_1_FWD_OPU_CUT;
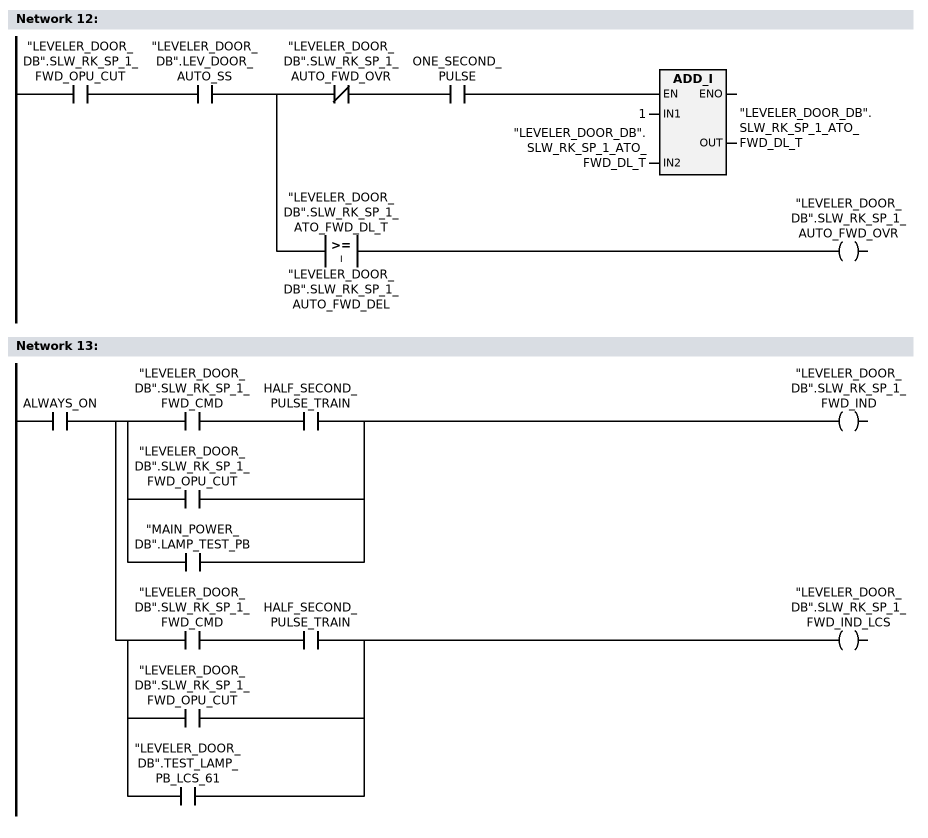
NETWORK
TITLE =
      A     "LEVELER_DOOR_DB".SLW_RK_SP_1_FWD_OPU_CUT;
      A     "LEVELER_DOOR_DB".LEV_DOOR_AUTO_SS;
      =     L 0.0;
      A     L 0.0;
      AN    "LEVELER_DOOR_DB".SLW_RK_SP_1_AUTO_FWD_OVR;
      A     "ONE_SECOND_PULSE";
      JNB   M006;
      L     1;
      L     "LEVELER_DOOR_DB".SLW_RK_SP_1_ATO_FWD_DL_T;
      +I;
      T     "LEVELER_DOOR_DB".SLW_RK_SP_1_ATO_FWD_DL_T;
M006: NOP   0;
      A     L 0.0;
      A(;
      L     "LEVELER_DOOR_DB".SLW_RK_SP_1_ATO_FWD_DL_T;
      L     "LEVELER_DOOR_DB".SLW_RK_SP_1_AUTO_FWD_DEL;
      >=I;
      );
      =     "LEVELER_DOOR_DB".SLW_RK_SP_1_AUTO_FWD_OVR;
NETWORK
TITLE =
      A     "ALWAYS_ON";
      =     L 0.0;
      A     L 0.0;
      A(;
      A     "LEVELER_DOOR_DB".SLW_RK_SP_1_FWD_CMD;
      A     "HALF_SECOND_PULSE_TRAIN";
      O     "LEVELER_DOOR_DB".SLW_RK_SP_1_FWD_OPU_CUT;
      O     "MAIN_POWER_DB".LAMP_TEST_PB;
      );
      =     "LEVELER_DOOR_DB".SLW_RK_SP_1_FWD_IND;
      A     L 0.0;
      A(;
      A     "LEVELER_DOOR_DB".SLW_RK_SP_1_FWD_CMD;
      A     "HALF_SECOND_PULSE_TRAIN";
      O     "LEVELER_DOOR_DB".SLW_RK_SP_1_FWD_OPU_CUT;
      O     "LEVELER_DOOR_DB".TEST_LAMP_PB_LCS_61;
      );
      =     "LEVELER_DOOR_DB".SLW_RK_SP_1_FWD_IND_LCS;
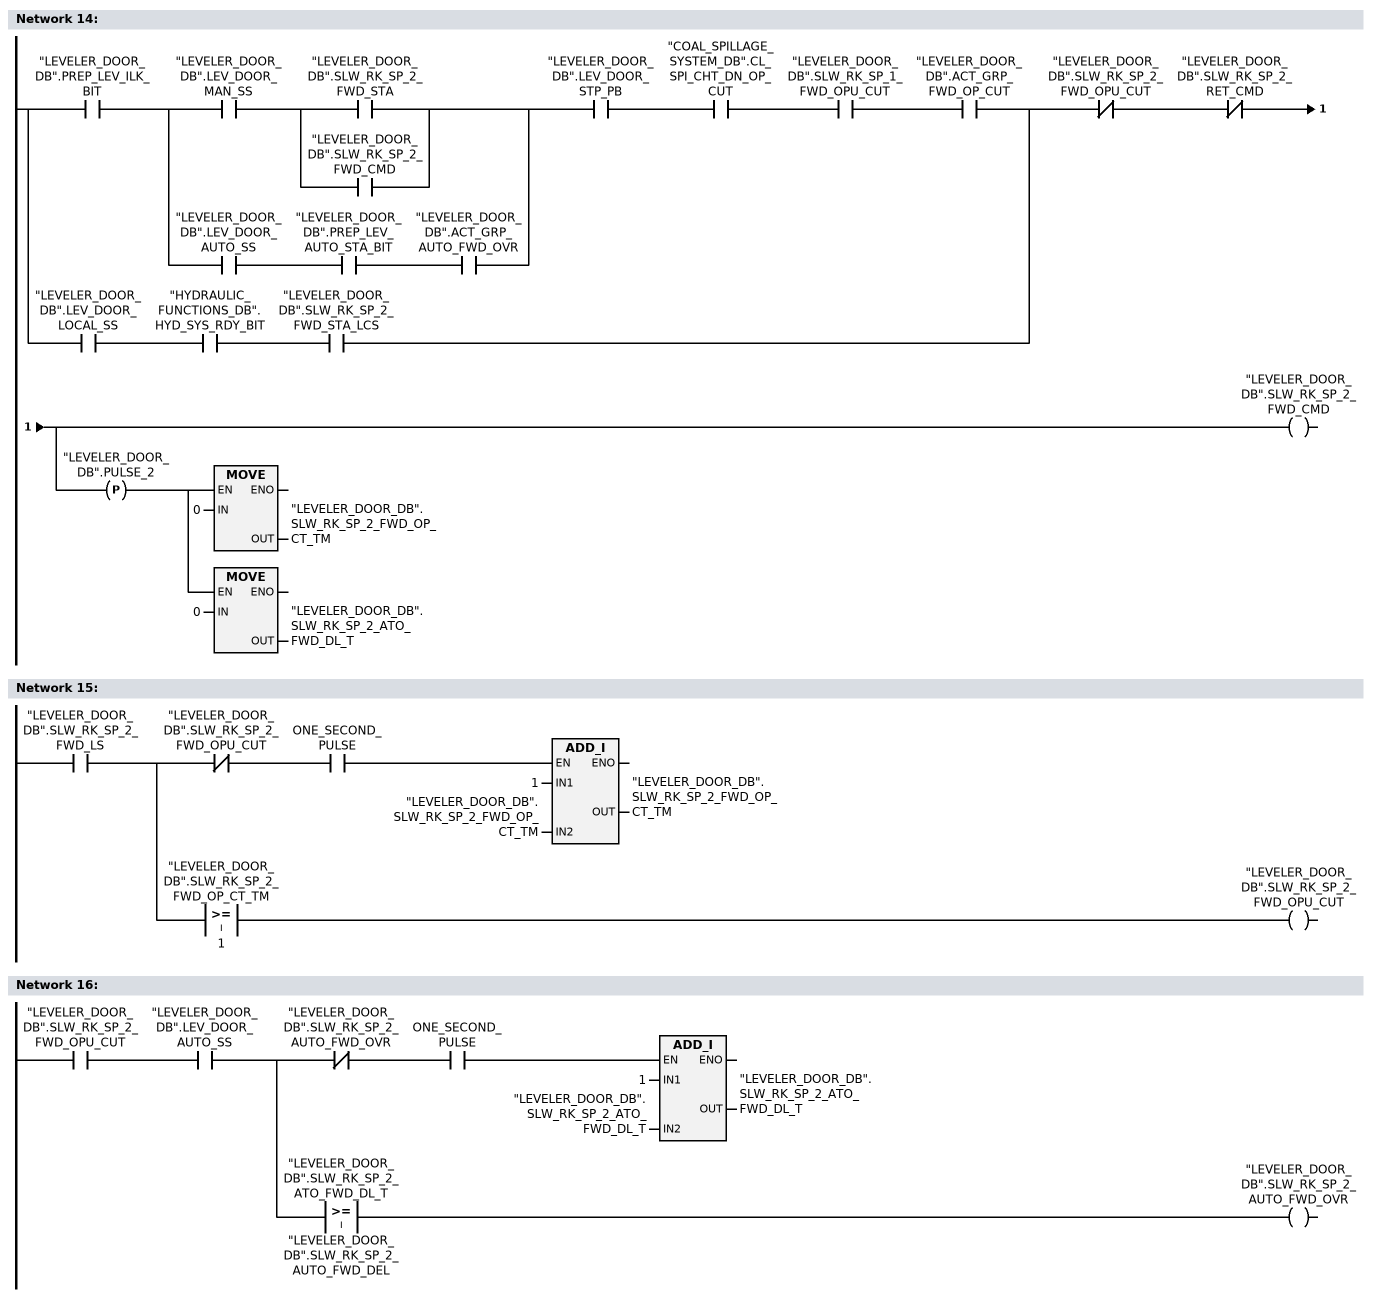
NETWORK
TITLE =
      A(;
      A     "LEVELER_DOOR_DB".PREP_LEV_ILK_BIT;
      A(;
      A     "LEVELER_DOOR_DB".LEV_DOOR_MAN_SS;
      A(;
      O     "LEVELER_DOOR_DB".SLW_RK_SP_2_FWD_STA;
      O     "LEVELER_DOOR_DB".SLW_RK_SP_2_FWD_CMD;
      );
      O;
      A     "LEVELER_DOOR_DB".LEV_DOOR_AUTO_SS;
      A     "LEVELER_DOOR_DB".PREP_LEV_AUTO_STA_BIT;
      A     "LEVELER_DOOR_DB".ACT_GRP_AUTO_FWD_OVR;
      );
      A     "LEVELER_DOOR_DB".LEV_DOOR_STP_PB;
      A     "COAL_SPILLAGE_SYSTEM_DB".CL_SPI_CHT_DN_OP_CUT;
      A     "LEVELER_DOOR_DB".SLW_RK_SP_1_FWD_OPU_CUT;
      A     "LEVELER_DOOR_DB".ACT_GRP_FWD_OP_CUT;
      O;
      A     "LEVELER_DOOR_DB".LEV_DOOR_LOCAL_SS;
      A     "HYDRAULIC_FUNCTIONS_DB".HYD_SYS_RDY_BIT;
      A     "LEVELER_DOOR_DB".SLW_RK_SP_2_FWD_STA_LCS;
      );
      AN    "LEVELER_DOOR_DB".SLW_RK_SP_2_FWD_OPU_CUT;
      AN    "LEVELER_DOOR_DB".SLW_RK_SP_2_RET_CMD;
      =     L 0.0;
      A     L 0.0;
      BLD   102;
      =     "LEVELER_DOOR_DB".SLW_RK_SP_2_FWD_CMD;
      A     L 0.0;
      FP    "LEVELER_DOOR_DB".PULSE_2;
      =     L 0.1;
      A     L 0.1;
      JNB   M007;
      L     0;
      T     "LEVELER_DOOR_DB".SLW_RK_SP_2_FWD_OP_CT_TM;
M007: NOP   0;
      A     L 0.1;
      JNB   M008;
      L     0;
      T     "LEVELER_DOOR_DB".SLW_RK_SP_2_ATO_FWD_DL_T;
M008: NOP   0;
NETWORK
TITLE =
      A     "LEVELER_DOOR_DB".SLW_RK_SP_2_FWD_LS;
      =     L 0.0;
      A     L 0.0;
      AN    "LEVELER_DOOR_DB".SLW_RK_SP_2_FWD_OPU_CUT;
      A     "ONE_SECOND_PULSE";
      JNB   M009;
      L     1;
      L     "LEVELER_DOOR_DB".SLW_RK_SP_2_FWD_OP_CT_TM;
      +I;
      T     "LEVELER_DOOR_DB".SLW_RK_SP_2_FWD_OP_CT_TM;
M009: NOP   0;
      A     L 0.0;
      A(;
      L     "LEVELER_DOOR_DB".SLW_RK_SP_2_FWD_OP_CT_TM;
      L     1;
      >=I;
      );
      =     "LEVELER_DOOR_DB".SLW_RK_SP_2_FWD_OPU_CUT;
NETWORK
TITLE =
      A     "LEVELER_DOOR_DB".SLW_RK_SP_2_FWD_OPU_CUT;
      A     "LEVELER_DOOR_DB".LEV_DOOR_AUTO_SS;
      =     L 0.0;
      A     L 0.0;
      AN    "LEVELER_DOOR_DB".SLW_RK_SP_2_AUTO_FWD_OVR;
      A     "ONE_SECOND_PULSE";
      JNB   M010;
      L     1;
      L     "LEVELER_DOOR_DB".SLW_RK_SP_2_ATO_FWD_DL_T;
      +I;
      T     "LEVELER_DOOR_DB".SLW_RK_SP_2_ATO_FWD_DL_T;
M010: NOP   0;
      A     L 0.0;
      A(;
      L     "LEVELER_DOOR_DB".SLW_RK_SP_2_ATO_FWD_DL_T;
      L     "LEVELER_DOOR_DB".SLW_RK_SP_2_AUTO_FWD_DEL;
      >=I;
      );
      =     "LEVELER_DOOR_DB".SLW_RK_SP_2_AUTO_FWD_OVR;
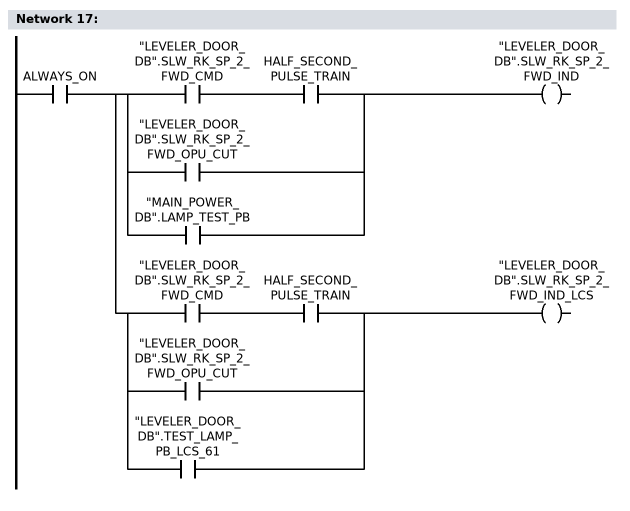
NETWORK
TITLE =
      A     "ALWAYS_ON";
      =     L 0.0;
      A     L 0.0;
      A(;
      A     "LEVELER_DOOR_DB".SLW_RK_SP_2_FWD_CMD;
      A     "HALF_SECOND_PULSE_TRAIN";
      O     "LEVELER_DOOR_DB".SLW_RK_SP_2_FWD_OPU_CUT;
      O     "MAIN_POWER_DB".LAMP_TEST_PB;
      );
      =     "LEVELER_DOOR_DB".SLW_RK_SP_2_FWD_IND;
      A     L 0.0;
      A(;
      A     "LEVELER_DOOR_DB".SLW_RK_SP_2_FWD_CMD;
      A     "HALF_SECOND_PULSE_TRAIN";
      O     "LEVELER_DOOR_DB".SLW_RK_SP_2_FWD_OPU_CUT;
      O     "LEVELER_DOOR_DB".TEST_LAMP_PB_LCS_61;
      );
      =     "LEVELER_DOOR_DB".SLW_RK_SP_2_FWD_IND_LCS;
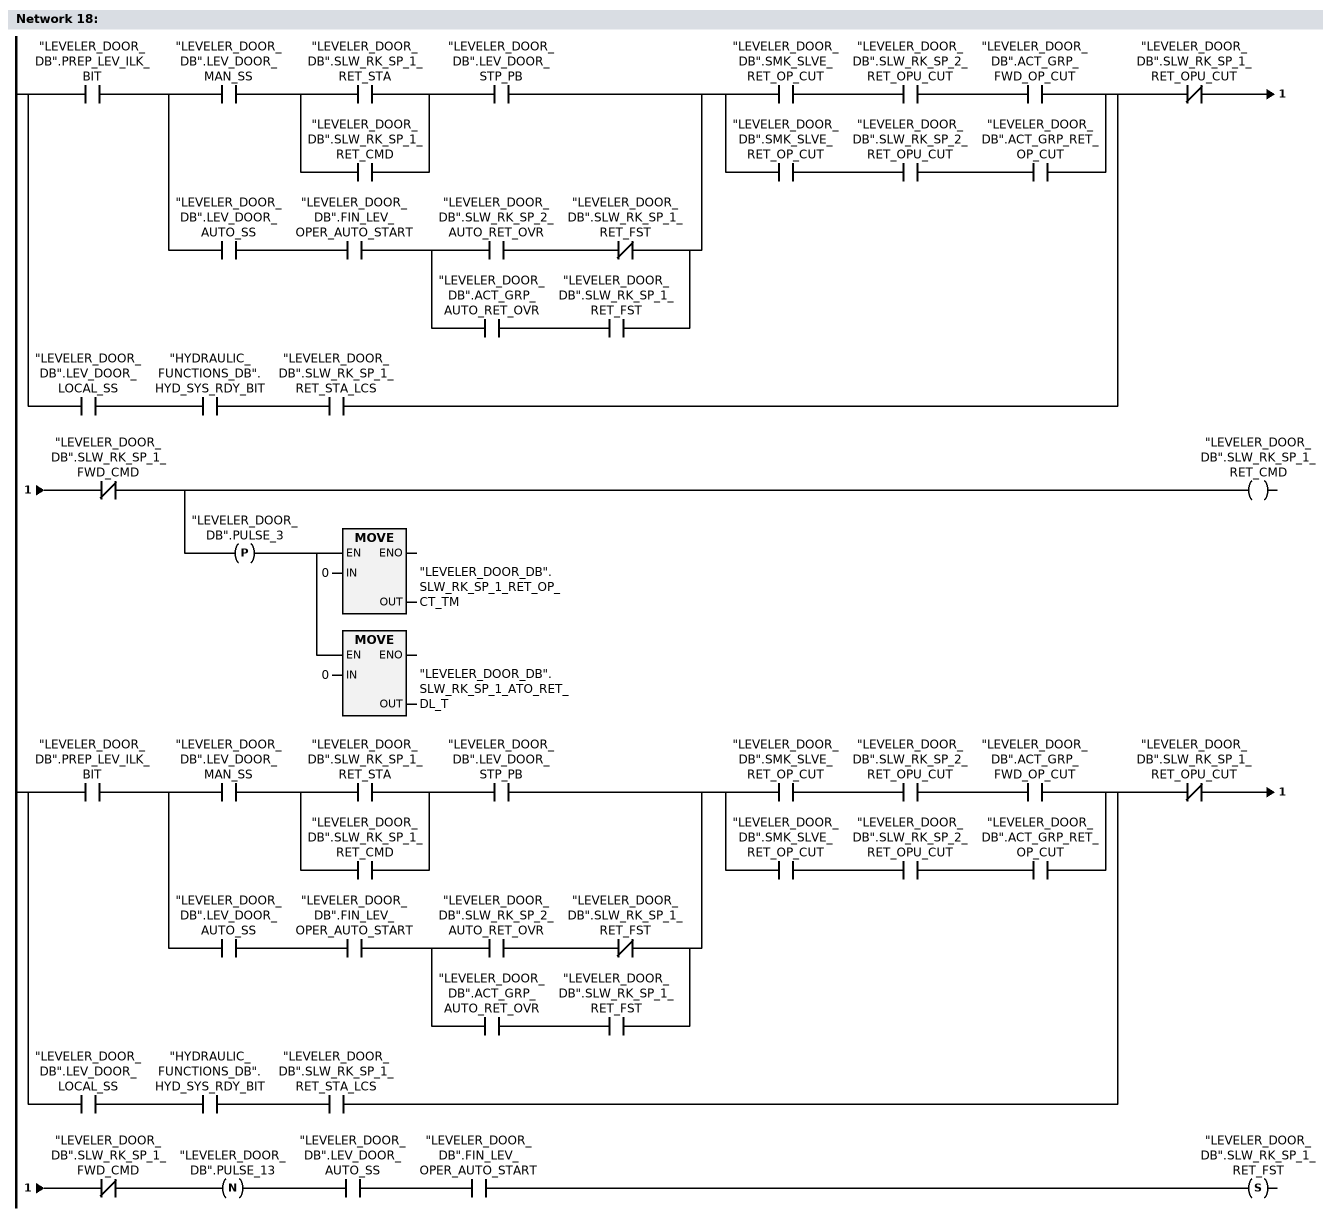
NETWORK
TITLE =
      A(;
      A     "LEVELER_DOOR_DB".PREP_LEV_ILK_BIT;
      A(;
      A     "LEVELER_DOOR_DB".LEV_DOOR_MAN_SS;
      A(;
      O     "LEVELER_DOOR_DB".SLW_RK_SP_1_RET_STA;
      O     "LEVELER_DOOR_DB".SLW_RK_SP_1_RET_CMD;
      );
      A     "LEVELER_DOOR_DB".LEV_DOOR_STP_PB;
      O;
      A     "LEVELER_DOOR_DB".LEV_DOOR_AUTO_SS;
      A     "LEVELER_DOOR_DB".FIN_LEV_OPER_AUTO_START;
      A(;
      A     "LEVELER_DOOR_DB".SLW_RK_SP_2_AUTO_RET_OVR;
      AN    "LEVELER_DOOR_DB".SLW_RK_SP_1_RET_FST;
      O;
      A     "LEVELER_DOOR_DB".ACT_GRP_AUTO_RET_OVR;
      A     "LEVELER_DOOR_DB".SLW_RK_SP_1_RET_FST;
      );
      );
      A(;
      A     "LEVELER_DOOR_DB".SMK_SLVE_RET_OP_CUT;
      A     "LEVELER_DOOR_DB".SLW_RK_SP_2_RET_OPU_CUT;
      A     "LEVELER_DOOR_DB".ACT_GRP_FWD_OP_CUT;
      O;
      A     "LEVELER_DOOR_DB".SMK_SLVE_RET_OP_CUT;
      A     "LEVELER_DOOR_DB".SLW_RK_SP_2_RET_OPU_CUT;
      A     "LEVELER_DOOR_DB".ACT_GRP_RET_OP_CUT;
      );
      O;
      A     "LEVELER_DOOR_DB".LEV_DOOR_LOCAL_SS;
      A     "HYDRAULIC_FUNCTIONS_DB".HYD_SYS_RDY_BIT;
      A     "LEVELER_DOOR_DB".SLW_RK_SP_1_RET_STA_LCS;
      );
      AN    "LEVELER_DOOR_DB".SLW_RK_SP_1_RET_OPU_CUT;
      AN    "LEVELER_DOOR_DB".SLW_RK_SP_1_FWD_CMD;
      =     L 0.0;
      A     L 0.0;
      BLD   102;
      =     "LEVELER_DOOR_DB".SLW_RK_SP_1_RET_CMD;
      A(;
      A     L 0.0;
      FN    "LEVELER_DOOR_DB".PULSE_13;
      );
      A     "LEVELER_DOOR_DB".LEV_DOOR_AUTO_SS;
      A     "LEVELER_DOOR_DB".FIN_LEV_OPER_AUTO_START;
      S     "LEVELER_DOOR_DB".SLW_RK_SP_1_RET_FST;
      A     L 0.0;
      FP    "LEVELER_DOOR_DB".PULSE_3;
      =     L 0.1;
      A     L 0.1;
      JNB   M011;
      L     0;
      T     "LEVELER_DOOR_DB".SLW_RK_SP_1_RET_OP_CT_TM;
M011: NOP   0;
      A     L 0.1;
      JNB   M012;
      L     0;
      T     "LEVELER_DOOR_DB".SLW_RK_SP_1_ATO_RET_DL_T;
M012: NOP   0;
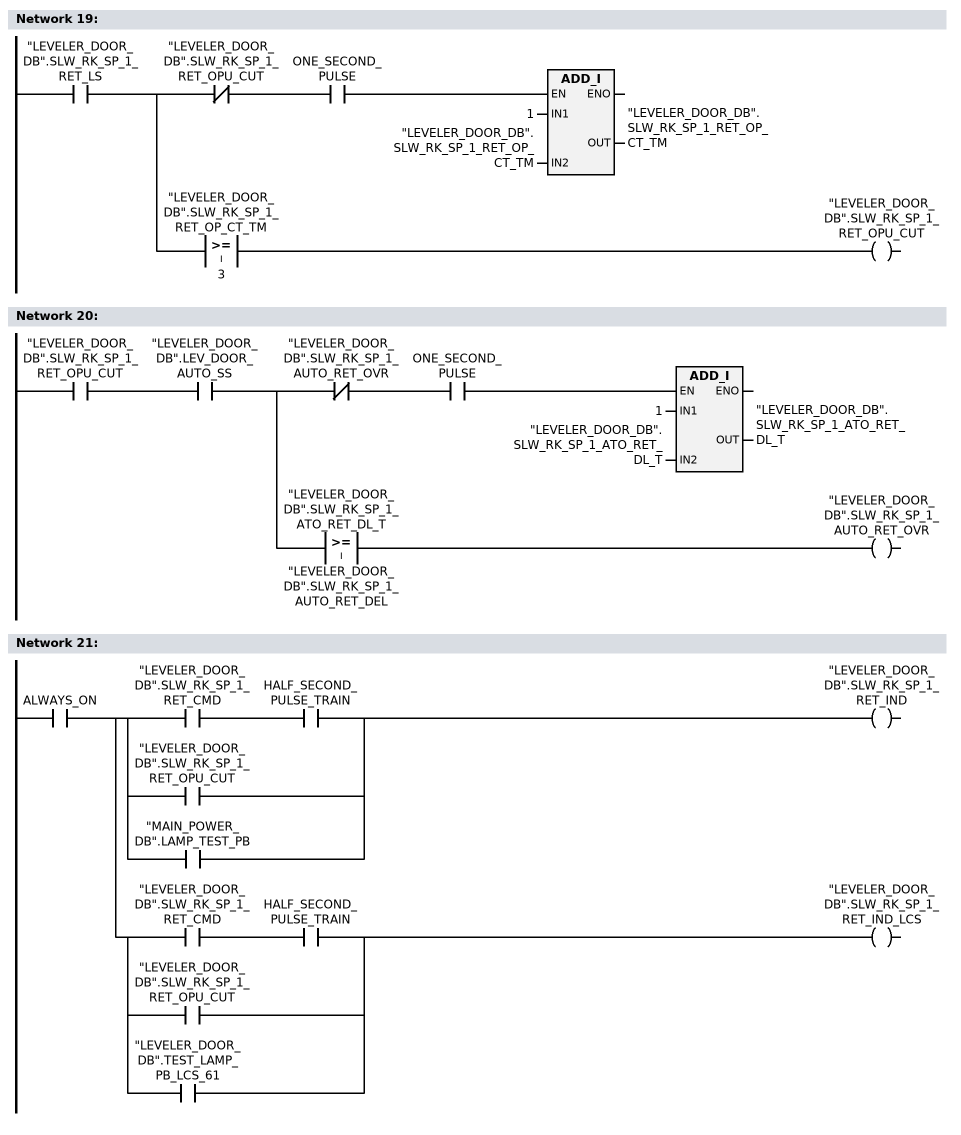
NETWORK
TITLE =
      A     "LEVELER_DOOR_DB".SLW_RK_SP_1_RET_LS;
      =     L 0.0;
      A     L 0.0;
      AN    "LEVELER_DOOR_DB".SLW_RK_SP_1_RET_OPU_CUT;
      A     "ONE_SECOND_PULSE";
      JNB   M013;
      L     1;
      L     "LEVELER_DOOR_DB".SLW_RK_SP_1_RET_OP_CT_TM;
      +I;
      T     "LEVELER_DOOR_DB".SLW_RK_SP_1_RET_OP_CT_TM;
M013: NOP   0;
      A     L 0.0;
      A(;
      L     "LEVELER_DOOR_DB".SLW_RK_SP_1_RET_OP_CT_TM;
      L     3;
      >=I;
      );
      =     "LEVELER_DOOR_DB".SLW_RK_SP_1_RET_OPU_CUT;
NETWORK
TITLE =
      A     "LEVELER_DOOR_DB".SLW_RK_SP_1_RET_OPU_CUT;
      A     "LEVELER_DOOR_DB".LEV_DOOR_AUTO_SS;
      =     L 0.0;
      A     L 0.0;
      AN    "LEVELER_DOOR_DB".SLW_RK_SP_1_AUTO_RET_OVR;
      A     "ONE_SECOND_PULSE";
      JNB   M014;
      L     1;
      L     "LEVELER_DOOR_DB".SLW_RK_SP_1_ATO_RET_DL_T;
      +I;
      T     "LEVELER_DOOR_DB".SLW_RK_SP_1_ATO_RET_DL_T;
M014: NOP   0;
      A     L 0.0;
      A(;
      L     "LEVELER_DOOR_DB".SLW_RK_SP_1_ATO_RET_DL_T;
      L     "LEVELER_DOOR_DB".SLW_RK_SP_1_AUTO_RET_DEL;
      >=I;
      );
      =     "LEVELER_DOOR_DB".SLW_RK_SP_1_AUTO_RET_OVR;
NETWORK
TITLE =
      A     "ALWAYS_ON";
      =     L 0.0;
      A     L 0.0;
      A(;
      A     "LEVELER_DOOR_DB".SLW_RK_SP_1_RET_CMD;
      A     "HALF_SECOND_PULSE_TRAIN";
      O     "LEVELER_DOOR_DB".SLW_RK_SP_1_RET_OPU_CUT;
      O     "MAIN_POWER_DB".LAMP_TEST_PB;
      );
      =     "LEVELER_DOOR_DB".SLW_RK_SP_1_RET_IND;
      A     L 0.0;
      A(;
      A     "LEVELER_DOOR_DB".SLW_RK_SP_1_RET_CMD;
      A     "HALF_SECOND_PULSE_TRAIN";
      O     "LEVELER_DOOR_DB".SLW_RK_SP_1_RET_OPU_CUT;
      O     "LEVELER_DOOR_DB".TEST_LAMP_PB_LCS_61;
      );
      =     "LEVELER_DOOR_DB".SLW_RK_SP_1_RET_IND_LCS;
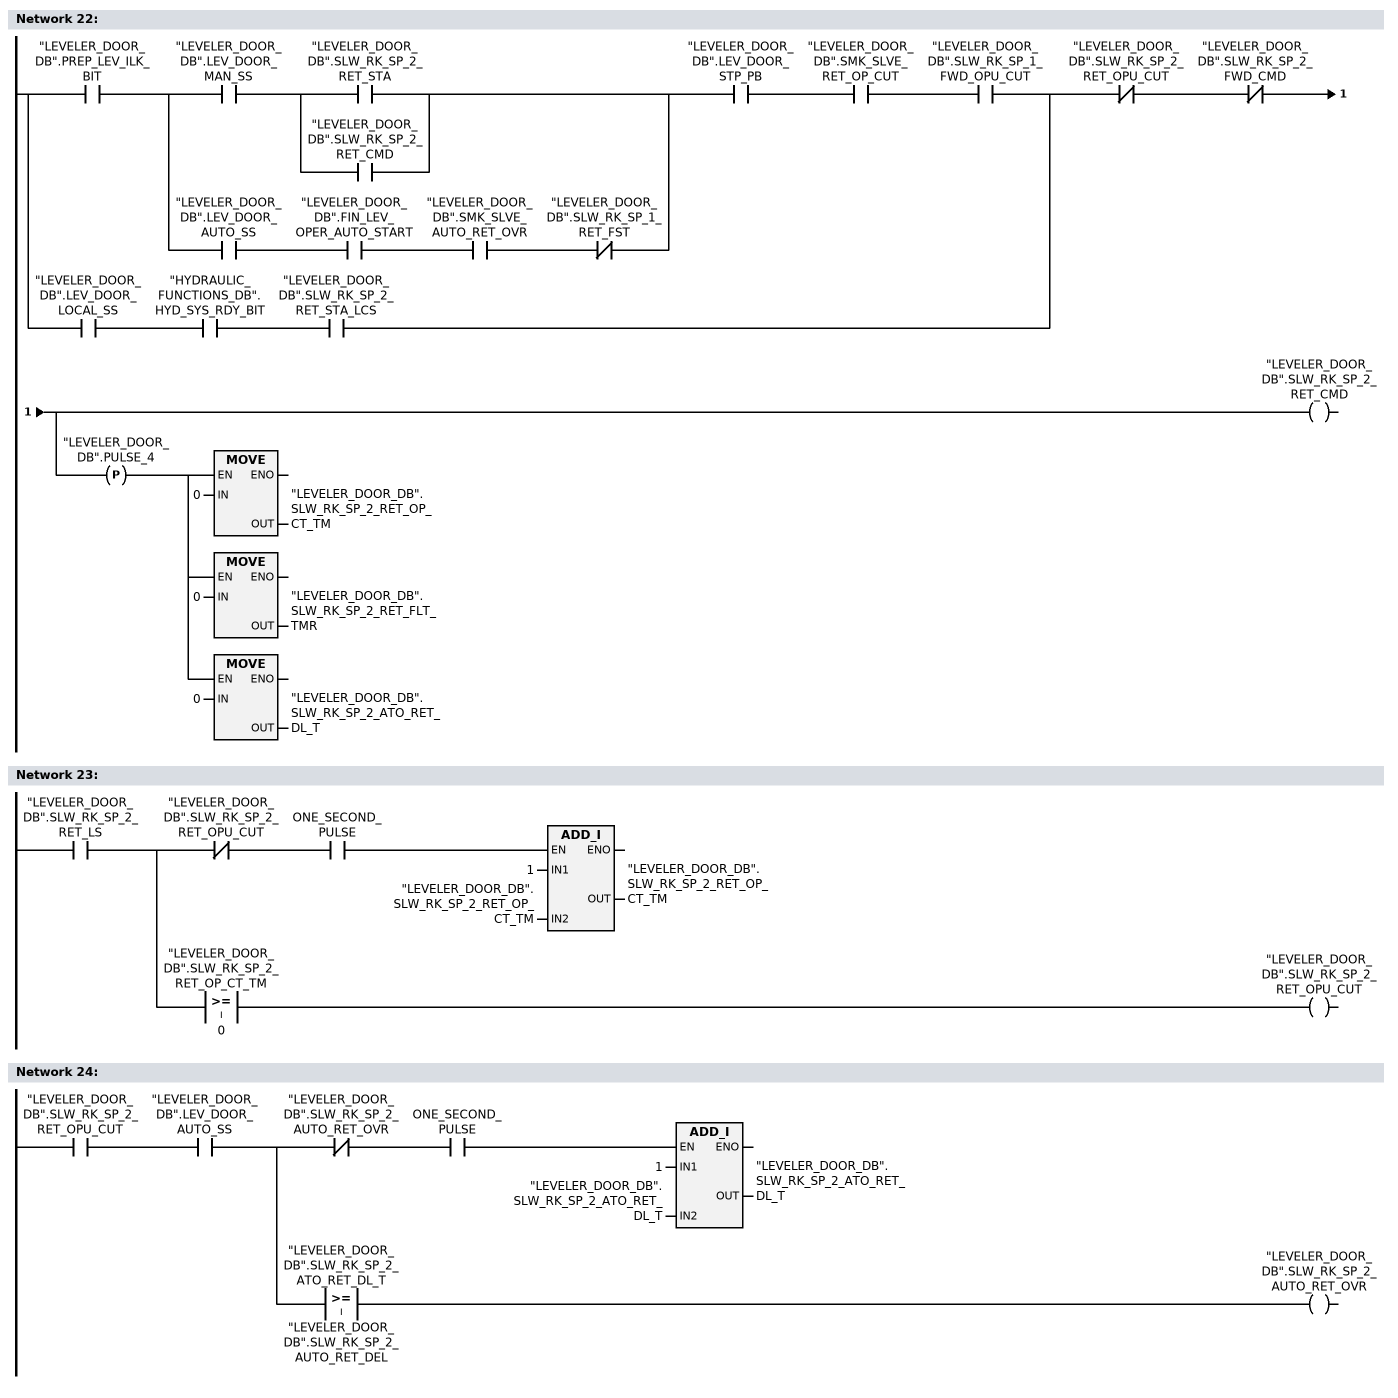
NETWORK
TITLE =
      A(;
      A     "LEVELER_DOOR_DB".PREP_LEV_ILK_BIT;
      A(;
      A     "LEVELER_DOOR_DB".LEV_DOOR_MAN_SS;
      A(;
      O     "LEVELER_DOOR_DB".SLW_RK_SP_2_RET_STA;
      O     "LEVELER_DOOR_DB".SLW_RK_SP_2_RET_CMD;
      );
      O;
      A     "LEVELER_DOOR_DB".LEV_DOOR_AUTO_SS;
      A     "LEVELER_DOOR_DB".FIN_LEV_OPER_AUTO_START;
      A     "LEVELER_DOOR_DB".SMK_SLVE_AUTO_RET_OVR;
      AN    "LEVELER_DOOR_DB".SLW_RK_SP_1_RET_FST;
      );
      A     "LEVELER_DOOR_DB".LEV_DOOR_STP_PB;
      A     "LEVELER_DOOR_DB".SMK_SLVE_RET_OP_CUT;
      A     "LEVELER_DOOR_DB".SLW_RK_SP_1_FWD_OPU_CUT;
      O;
      A     "LEVELER_DOOR_DB".LEV_DOOR_LOCAL_SS;
      A     "HYDRAULIC_FUNCTIONS_DB".HYD_SYS_RDY_BIT;
      A     "LEVELER_DOOR_DB".SLW_RK_SP_2_RET_STA_LCS;
      );
      AN    "LEVELER_DOOR_DB".SLW_RK_SP_2_RET_OPU_CUT;
      AN    "LEVELER_DOOR_DB".SLW_RK_SP_2_FWD_CMD;
      =     L 0.0;
      A     L 0.0;
      BLD   102;
      =     "LEVELER_DOOR_DB".SLW_RK_SP_2_RET_CMD;
      A     L 0.0;
      FP    "LEVELER_DOOR_DB".PULSE_4;
      =     L 0.1;
      A     L 0.1;
      JNB   M015;
      L     0;
      T     "LEVELER_DOOR_DB".SLW_RK_SP_2_RET_OP_CT_TM;
M015: NOP   0;
      A     L 0.1;
      JNB   M016;
      L     0;
      T     "LEVELER_DOOR_DB".SLW_RK_SP_2_RET_FLT_TMR;
M016: NOP   0;
      A     L 0.1;
      JNB   M017;
      L     0;
      T     "LEVELER_DOOR_DB".SLW_RK_SP_2_ATO_RET_DL_T;
M017: NOP   0;
NETWORK
TITLE =
      A     "LEVELER_DOOR_DB".SLW_RK_SP_2_RET_LS;
      =     L 0.0;
      A     L 0.0;
      AN    "LEVELER_DOOR_DB".SLW_RK_SP_2_RET_OPU_CUT;
      A     "ONE_SECOND_PULSE";
      JNB   M018;
      L     1;
      L     "LEVELER_DOOR_DB".SLW_RK_SP_2_RET_OP_CT_TM;
      +I;
      T     "LEVELER_DOOR_DB".SLW_RK_SP_2_RET_OP_CT_TM;
M018: NOP   0;
      A     L 0.0;
      A(;
      L     "LEVELER_DOOR_DB".SLW_RK_SP_2_RET_OP_CT_TM;
      L     0;
      >=I;
      );
      =     "LEVELER_DOOR_DB".SLW_RK_SP_2_RET_OPU_CUT;
NETWORK
TITLE =
      A     "LEVELER_DOOR_DB".SLW_RK_SP_2_RET_OPU_CUT;
      A     "LEVELER_DOOR_DB".LEV_DOOR_AUTO_SS;
      =     L 0.0;
      A     L 0.0;
      AN    "LEVELER_DOOR_DB".SLW_RK_SP_2_AUTO_RET_OVR;
      A     "ONE_SECOND_PULSE";
      JNB   M019;
      L     1;
      L     "LEVELER_DOOR_DB".SLW_RK_SP_2_ATO_RET_DL_T;
      +I;
      T     "LEVELER_DOOR_DB".SLW_RK_SP_2_ATO_RET_DL_T;
M019: NOP   0;
      A     L 0.0;
      A(;
      L     "LEVELER_DOOR_DB".SLW_RK_SP_2_ATO_RET_DL_T;
      L     "LEVELER_DOOR_DB".SLW_RK_SP_2_AUTO_RET_DEL;
      >=I;
      );
      =     "LEVELER_DOOR_DB".SLW_RK_SP_2_AUTO_RET_OVR;
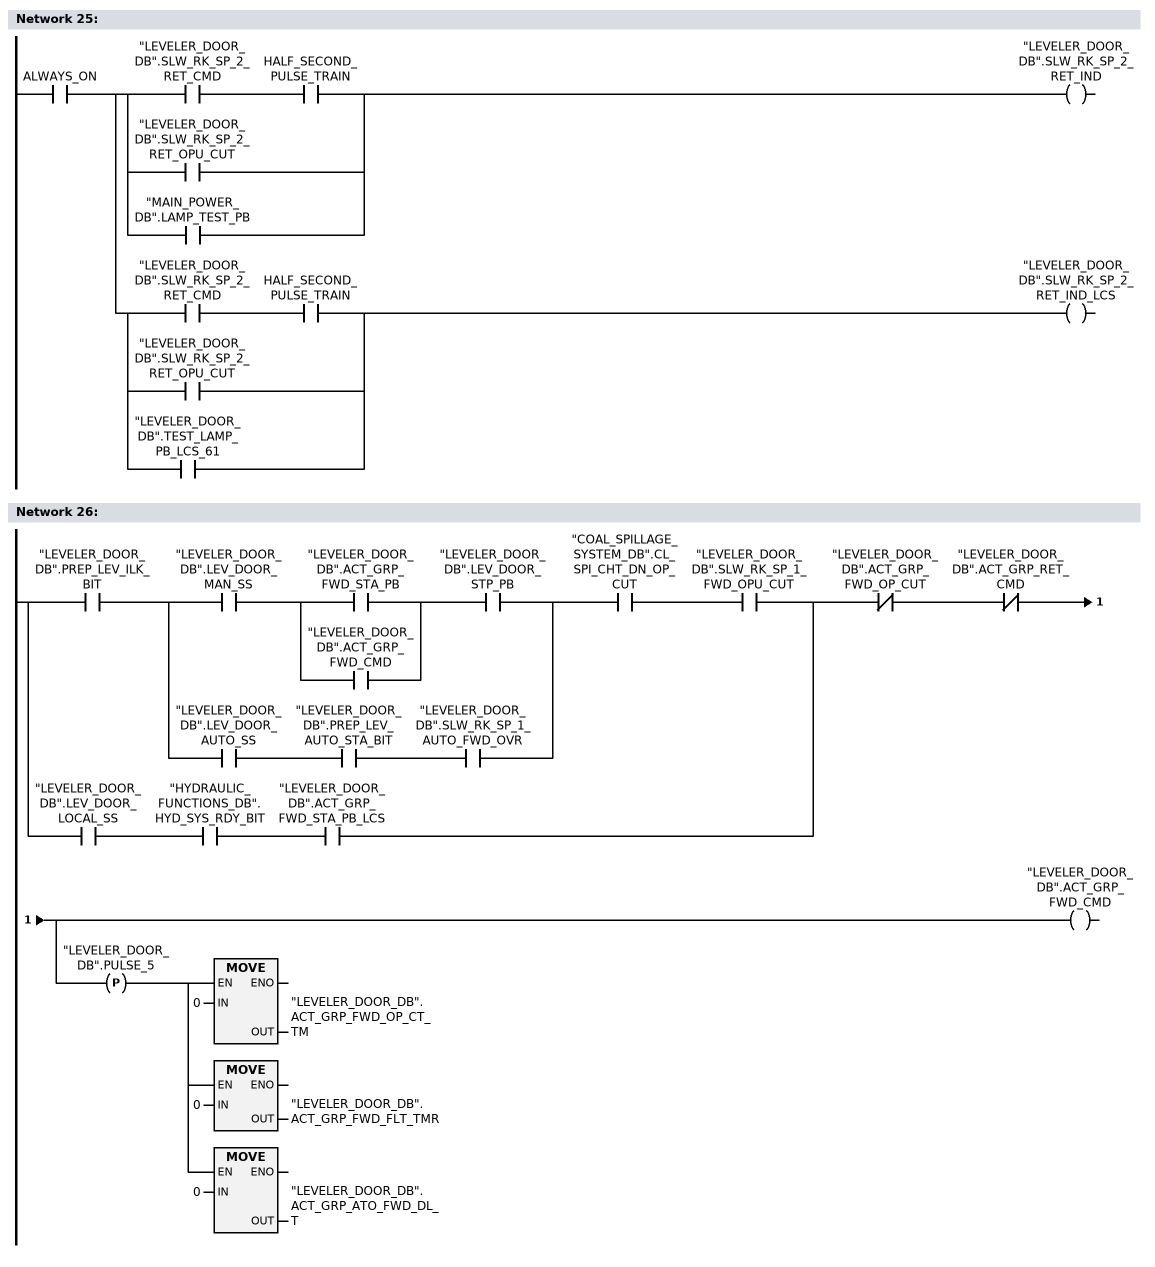
NETWORK
TITLE =
      A     "ALWAYS_ON";
      =     L 0.0;
      A     L 0.0;
      A(;
      A     "LEVELER_DOOR_DB".SLW_RK_SP_2_RET_CMD;
      A     "HALF_SECOND_PULSE_TRAIN";
      O     "LEVELER_DOOR_DB".SLW_RK_SP_2_RET_OPU_CUT;
      O     "MAIN_POWER_DB".LAMP_TEST_PB;
      );
      =     "LEVELER_DOOR_DB".SLW_RK_SP_2_RET_IND;
      A     L 0.0;
      A(;
      A     "LEVELER_DOOR_DB".SLW_RK_SP_2_RET_CMD;
      A     "HALF_SECOND_PULSE_TRAIN";
      O     "LEVELER_DOOR_DB".SLW_RK_SP_2_RET_OPU_CUT;
      O     "LEVELER_DOOR_DB".TEST_LAMP_PB_LCS_61;
      );
      =     "LEVELER_DOOR_DB".SLW_RK_SP_2_RET_IND_LCS;
NETWORK
TITLE =
      A(;
      A     "LEVELER_DOOR_DB".PREP_LEV_ILK_BIT;
      A(;
      A     "LEVELER_DOOR_DB".LEV_DOOR_MAN_SS;
      A(;
      O     "LEVELER_DOOR_DB".ACT_GRP_FWD_STA_PB;
      O     "LEVELER_DOOR_DB".ACT_GRP_FWD_CMD;
      );
      A     "LEVELER_DOOR_DB".LEV_DOOR_STP_PB;
      O;
      A     "LEVELER_DOOR_DB".LEV_DOOR_AUTO_SS;
      A     "LEVELER_DOOR_DB".PREP_LEV_AUTO_STA_BIT;
      A     "LEVELER_DOOR_DB".SLW_RK_SP_1_AUTO_FWD_OVR;
      );
      A     "COAL_SPILLAGE_SYSTEM_DB".CL_SPI_CHT_DN_OP_CUT;
      A     "LEVELER_DOOR_DB".SLW_RK_SP_1_FWD_OPU_CUT;
      O;
      A     "LEVELER_DOOR_DB".LEV_DOOR_LOCAL_SS;
      A     "HYDRAULIC_FUNCTIONS_DB".HYD_SYS_RDY_BIT;
      A     "LEVELER_DOOR_DB".ACT_GRP_FWD_STA_PB_LCS;
      );
      AN    "LEVELER_DOOR_DB".ACT_GRP_FWD_OP_CUT;
      AN    "LEVELER_DOOR_DB".ACT_GRP_RET_CMD;
      =     L 0.0;
      A     L 0.0;
      BLD   102;
      =     "LEVELER_DOOR_DB".ACT_GRP_FWD_CMD;
      A     L 0.0;
      FP    "LEVELER_DOOR_DB".PULSE_5;
      =     L 0.1;
      A     L 0.1;
      JNB   M020;
      L     0;
      T     "LEVELER_DOOR_DB".ACT_GRP_FWD_OP_CT_TM;
M020: NOP   0;
      A     L 0.1;
      JNB   M021;
      L     0;
      T     "LEVELER_DOOR_DB".ACT_GRP_FWD_FLT_TMR;
M021: NOP   0;
      A     L 0.1;
      JNB   M022;
      L     0;
      T     "LEVELER_DOOR_DB".ACT_GRP_ATO_FWD_DL_T;
M022: NOP   0;
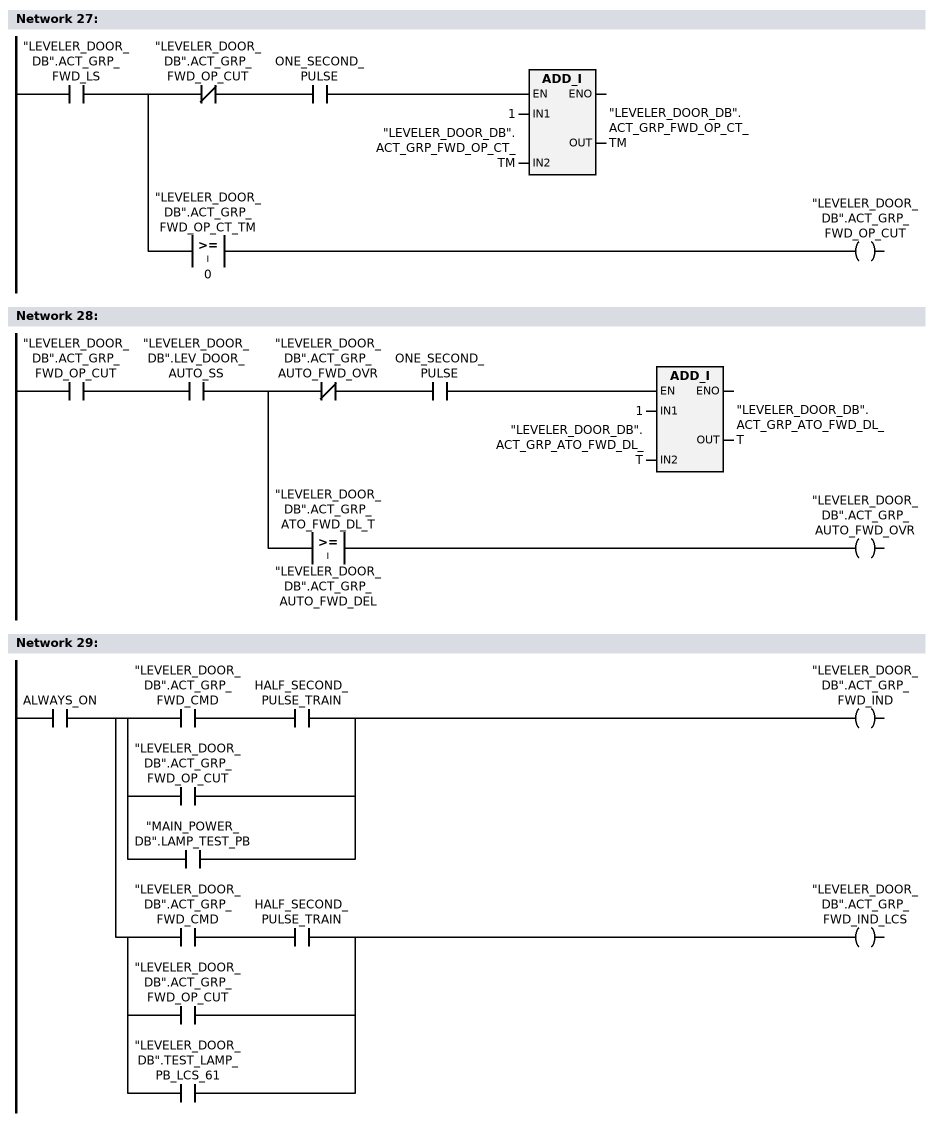
NETWORK
TITLE =
      A     "LEVELER_DOOR_DB".ACT_GRP_FWD_LS;
      =     L 0.0;
      A     L 0.0;
      AN    "LEVELER_DOOR_DB".ACT_GRP_FWD_OP_CUT;
      A     "ONE_SECOND_PULSE";
      JNB   M023;
      L     1;
      L     "LEVELER_DOOR_DB".ACT_GRP_FWD_OP_CT_TM;
      +I;
      T     "LEVELER_DOOR_DB".ACT_GRP_FWD_OP_CT_TM;
M023: NOP   0;
      A     L 0.0;
      A(;
      L     "LEVELER_DOOR_DB".ACT_GRP_FWD_OP_CT_TM;
      L     0;
      >=I;
      );
      =     "LEVELER_DOOR_DB".ACT_GRP_FWD_OP_CUT;
NETWORK
TITLE =
      A     "LEVELER_DOOR_DB".ACT_GRP_FWD_OP_CUT;
      A     "LEVELER_DOOR_DB".LEV_DOOR_AUTO_SS;
      =     L 0.0;
      A     L 0.0;
      AN    "LEVELER_DOOR_DB".ACT_GRP_AUTO_FWD_OVR;
      A     "ONE_SECOND_PULSE";
      JNB   M024;
      L     1;
      L     "LEVELER_DOOR_DB".ACT_GRP_ATO_FWD_DL_T;
      +I;
      T     "LEVELER_DOOR_DB".ACT_GRP_ATO_FWD_DL_T;
M024: NOP   0;
      A     L 0.0;
      A(;
      L     "LEVELER_DOOR_DB".ACT_GRP_ATO_FWD_DL_T;
      L     "LEVELER_DOOR_DB".ACT_GRP_AUTO_FWD_DEL;
      >=I;
      );
      =     "LEVELER_DOOR_DB".ACT_GRP_AUTO_FWD_OVR;
NETWORK
TITLE =
      A     "ALWAYS_ON";
      =     L 0.0;
      A     L 0.0;
      A(;
      A     "LEVELER_DOOR_DB".ACT_GRP_FWD_CMD;
      A     "HALF_SECOND_PULSE_TRAIN";
      O     "LEVELER_DOOR_DB".ACT_GRP_FWD_OP_CUT;
      O     "MAIN_POWER_DB".LAMP_TEST_PB;
      );
      =     "LEVELER_DOOR_DB".ACT_GRP_FWD_IND;
      A     L 0.0;
      A(;
      A     "LEVELER_DOOR_DB".ACT_GRP_FWD_CMD;
      A     "HALF_SECOND_PULSE_TRAIN";
      O     "LEVELER_DOOR_DB".ACT_GRP_FWD_OP_CUT;
      O     "LEVELER_DOOR_DB".TEST_LAMP_PB_LCS_61;
      );
      =     "LEVELER_DOOR_DB".ACT_GRP_FWD_IND_LCS;
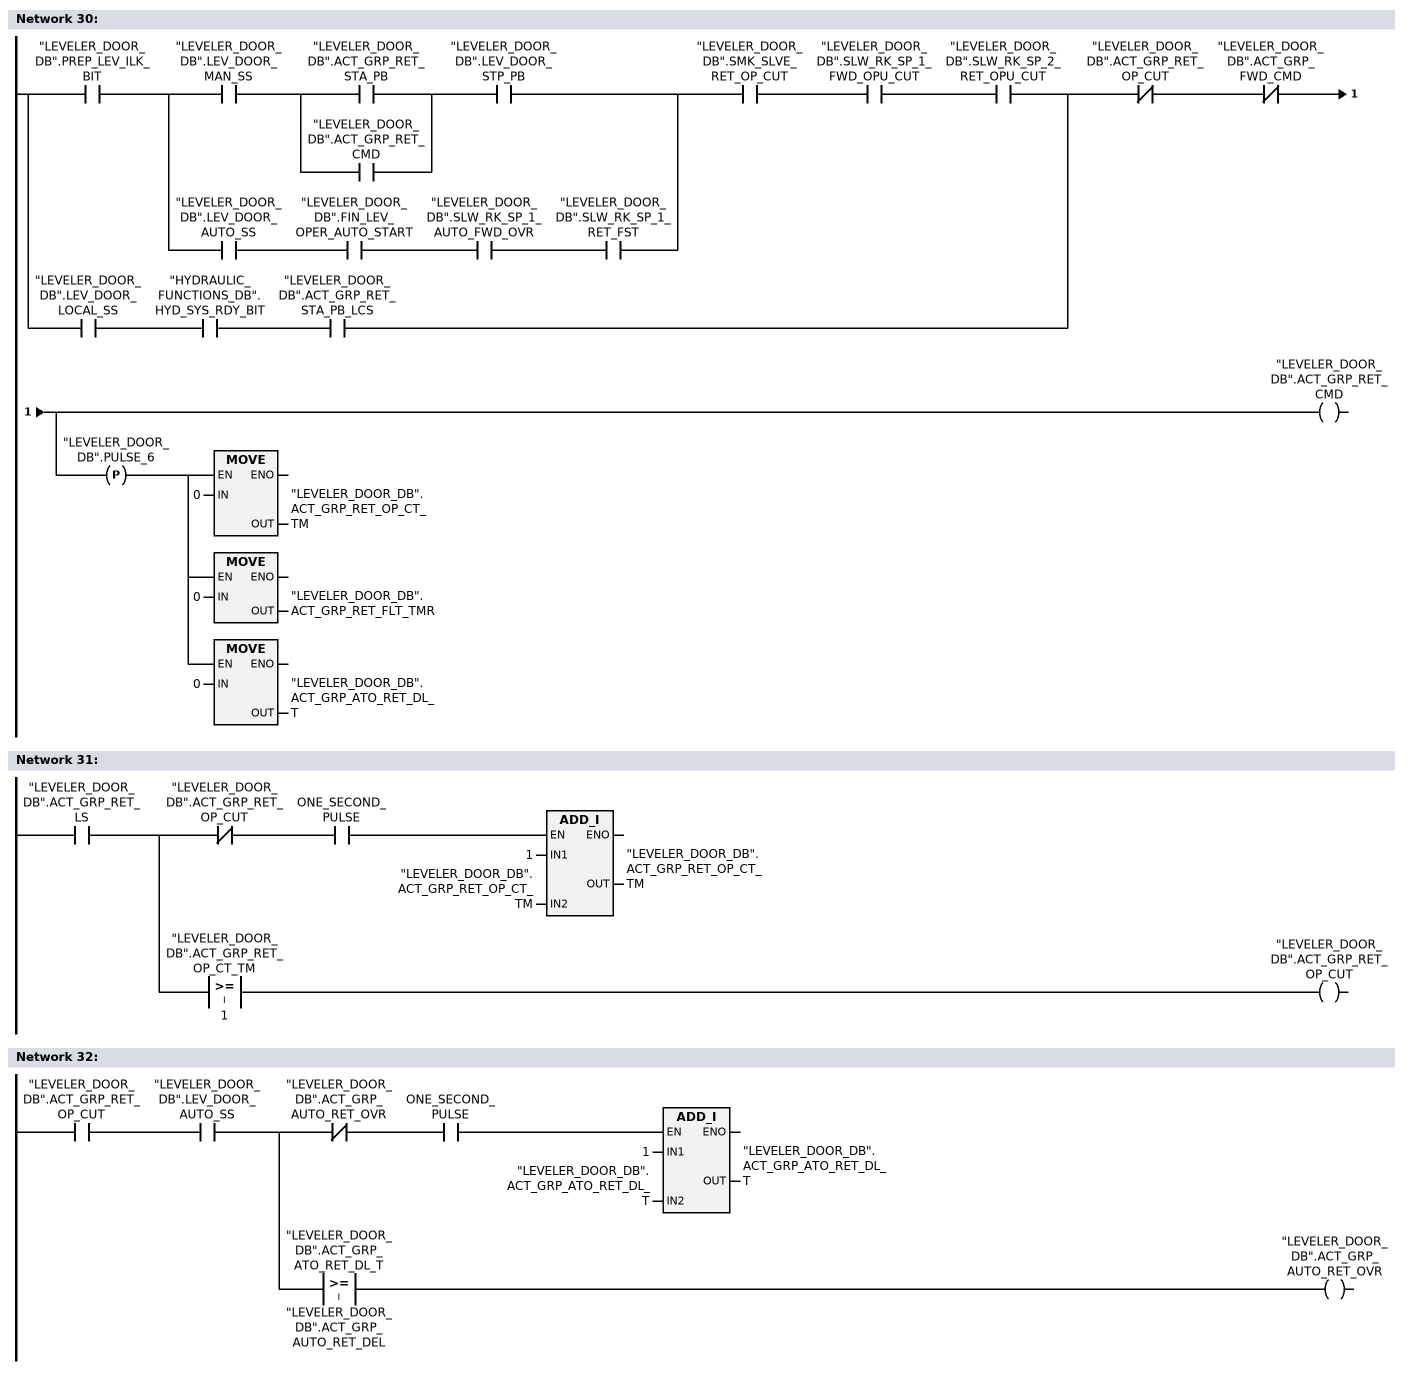
NETWORK
TITLE =
      A(;
      A     "LEVELER_DOOR_DB".PREP_LEV_ILK_BIT;
      A(;
      A     "LEVELER_DOOR_DB".LEV_DOOR_MAN_SS;
      A(;
      O     "LEVELER_DOOR_DB".ACT_GRP_RET_STA_PB;
      O     "LEVELER_DOOR_DB".ACT_GRP_RET_CMD;
      );
      A     "LEVELER_DOOR_DB".LEV_DOOR_STP_PB;
      O;
      A     "LEVELER_DOOR_DB".LEV_DOOR_AUTO_SS;
      A     "LEVELER_DOOR_DB".FIN_LEV_OPER_AUTO_START;
      A     "LEVELER_DOOR_DB".SLW_RK_SP_1_AUTO_FWD_OVR;
      A     "LEVELER_DOOR_DB".SLW_RK_SP_1_RET_FST;
      );
      A     "LEVELER_DOOR_DB".SMK_SLVE_RET_OP_CUT;
      A     "LEVELER_DOOR_DB".SLW_RK_SP_1_FWD_OPU_CUT;
      A     "LEVELER_DOOR_DB".SLW_RK_SP_2_RET_OPU_CUT;
      O;
      A     "LEVELER_DOOR_DB".LEV_DOOR_LOCAL_SS;
      A     "HYDRAULIC_FUNCTIONS_DB".HYD_SYS_RDY_BIT;
      A     "LEVELER_DOOR_DB".ACT_GRP_RET_STA_PB_LCS;
      );
      AN    "LEVELER_DOOR_DB".ACT_GRP_RET_OP_CUT;
      AN    "LEVELER_DOOR_DB".ACT_GRP_FWD_CMD;
      =     L 0.0;
      A     L 0.0;
      BLD   102;
      =     "LEVELER_DOOR_DB".ACT_GRP_RET_CMD;
      A     L 0.0;
      FP    "LEVELER_DOOR_DB".PULSE_6;
      =     L 0.1;
      A     L 0.1;
      JNB   M025;
      L     0;
      T     "LEVELER_DOOR_DB".ACT_GRP_RET_OP_CT_TM;
M025: NOP   0;
      A     L 0.1;
      JNB   M026;
      L     0;
      T     "LEVELER_DOOR_DB".ACT_GRP_RET_FLT_TMR;
M026: NOP   0;
      A     L 0.1;
      JNB   M027;
      L     0;
      T     "LEVELER_DOOR_DB".ACT_GRP_ATO_RET_DL_T;
M027: NOP   0;
NETWORK
TITLE =
      A     "LEVELER_DOOR_DB".ACT_GRP_RET_LS;
      =     L 0.0;
      A     L 0.0;
      AN    "LEVELER_DOOR_DB".ACT_GRP_RET_OP_CUT;
      A     "ONE_SECOND_PULSE";
      JNB   M028;
      L     1;
      L     "LEVELER_DOOR_DB".ACT_GRP_RET_OP_CT_TM;
      +I;
      T     "LEVELER_DOOR_DB".ACT_GRP_RET_OP_CT_TM;
M028: NOP   0;
      A     L 0.0;
      A(;
      L     "LEVELER_DOOR_DB".ACT_GRP_RET_OP_CT_TM;
      L     1;
      >=I;
      );
      =     "LEVELER_DOOR_DB".ACT_GRP_RET_OP_CUT;
NETWORK
TITLE =
      A     "LEVELER_DOOR_DB".ACT_GRP_RET_OP_CUT;
      A     "LEVELER_DOOR_DB".LEV_DOOR_AUTO_SS;
      =     L 0.0;
      A     L 0.0;
      AN    "LEVELER_DOOR_DB".ACT_GRP_AUTO_RET_OVR;
      A     "ONE_SECOND_PULSE";
      JNB   M029;
      L     1;
      L     "LEVELER_DOOR_DB".ACT_GRP_ATO_RET_DL_T;
      +I;
      T     "LEVELER_DOOR_DB".ACT_GRP_ATO_RET_DL_T;
M029: NOP   0;
      A     L 0.0;
      A(;
      L     "LEVELER_DOOR_DB".ACT_GRP_ATO_RET_DL_T;
      L     "LEVELER_DOOR_DB".ACT_GRP_AUTO_RET_DEL;
      >=I;
      );
      =     "LEVELER_DOOR_DB".ACT_GRP_AUTO_RET_OVR;
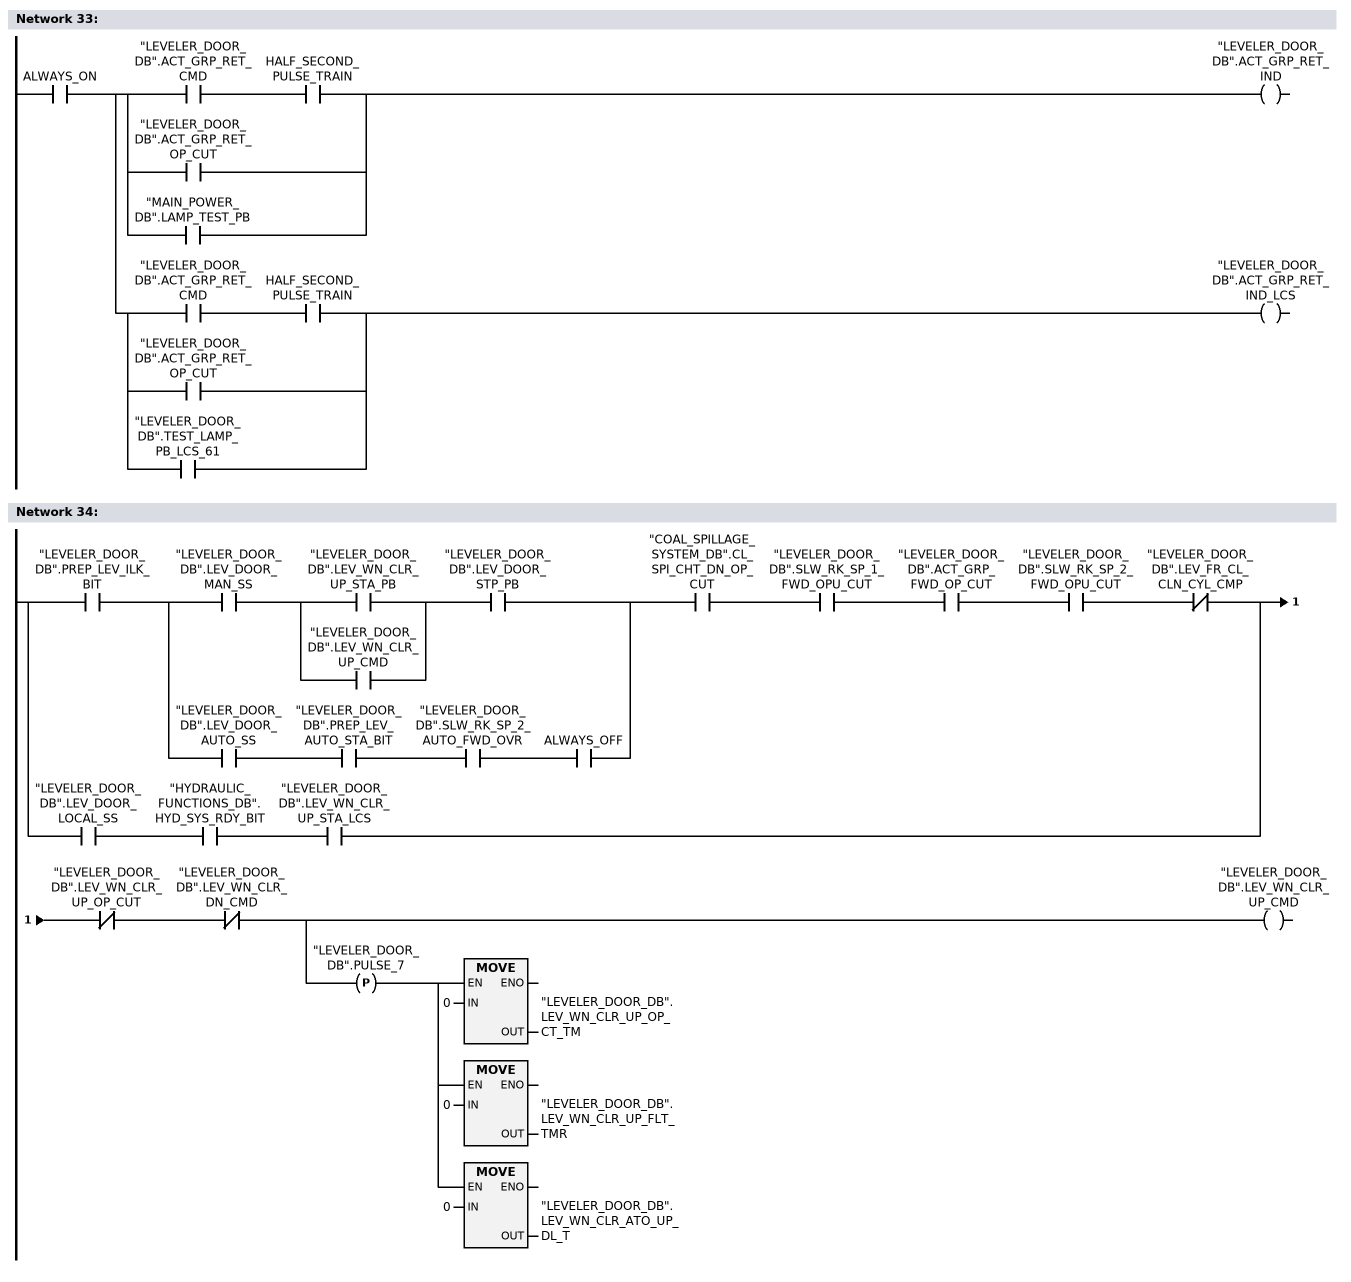
NETWORK
TITLE =
      A     "ALWAYS_ON";
      =     L 0.0;
      A     L 0.0;
      A(;
      A     "LEVELER_DOOR_DB".ACT_GRP_RET_CMD;
      A     "HALF_SECOND_PULSE_TRAIN";
      O     "LEVELER_DOOR_DB".ACT_GRP_RET_OP_CUT;
      O     "MAIN_POWER_DB".LAMP_TEST_PB;
      );
      =     "LEVELER_DOOR_DB".ACT_GRP_RET_IND;
      A     L 0.0;
      A(;
      A     "LEVELER_DOOR_DB".ACT_GRP_RET_CMD;
      A     "HALF_SECOND_PULSE_TRAIN";
      O     "LEVELER_DOOR_DB".ACT_GRP_RET_OP_CUT;
      O     "LEVELER_DOOR_DB".TEST_LAMP_PB_LCS_61;
      );
      =     "LEVELER_DOOR_DB".ACT_GRP_RET_IND_LCS;
NETWORK
TITLE =
      A(;
      A     "LEVELER_DOOR_DB".PREP_LEV_ILK_BIT;
      A(;
      A     "LEVELER_DOOR_DB".LEV_DOOR_MAN_SS;
      A(;
      O     "LEVELER_DOOR_DB".LEV_WN_CLR_UP_STA_PB;
      O     "LEVELER_DOOR_DB".LEV_WN_CLR_UP_CMD;
      );
      A     "LEVELER_DOOR_DB".LEV_DOOR_STP_PB;
      O;
      A     "LEVELER_DOOR_DB".LEV_DOOR_AUTO_SS;
      A     "LEVELER_DOOR_DB".PREP_LEV_AUTO_STA_BIT;
      A     "LEVELER_DOOR_DB".SLW_RK_SP_2_AUTO_FWD_OVR;
      A     "ALWAYS_OFF";
      );
      A     "COAL_SPILLAGE_SYSTEM_DB".CL_SPI_CHT_DN_OP_CUT;
      A     "LEVELER_DOOR_DB".SLW_RK_SP_1_FWD_OPU_CUT;
      A     "LEVELER_DOOR_DB".ACT_GRP_FWD_OP_CUT;
      A     "LEVELER_DOOR_DB".SLW_RK_SP_2_FWD_OPU_CUT;
      AN    "LEVELER_DOOR_DB".LEV_FR_CL_CLN_CYL_CMP;
      O;
      A     "LEVELER_DOOR_DB".LEV_DOOR_LOCAL_SS;
      A     "HYDRAULIC_FUNCTIONS_DB".HYD_SYS_RDY_BIT;
      A     "LEVELER_DOOR_DB".LEV_WN_CLR_UP_STA_LCS;
      );
      AN    "LEVELER_DOOR_DB".LEV_WN_CLR_UP_OP_CUT;
      AN    "LEVELER_DOOR_DB".LEV_WN_CLR_DN_CMD;
      =     L 0.0;
      A     L 0.0;
      BLD   102;
      =     "LEVELER_DOOR_DB".LEV_WN_CLR_UP_CMD;
      A     L 0.0;
      FP    "LEVELER_DOOR_DB".PULSE_7;
      =     L 0.1;
      A     L 0.1;
      JNB   M030;
      L     0;
      T     "LEVELER_DOOR_DB".LEV_WN_CLR_UP_OP_CT_TM;
M030: NOP   0;
      A     L 0.1;
      JNB   M031;
      L     0;
      T     "LEVELER_DOOR_DB".LEV_WN_CLR_UP_FLT_TMR;
M031: NOP   0;
      A     L 0.1;
      JNB   M032;
      L     0;
      T     "LEVELER_DOOR_DB".LEV_WN_CLR_ATO_UP_DL_T;
M032: NOP   0;
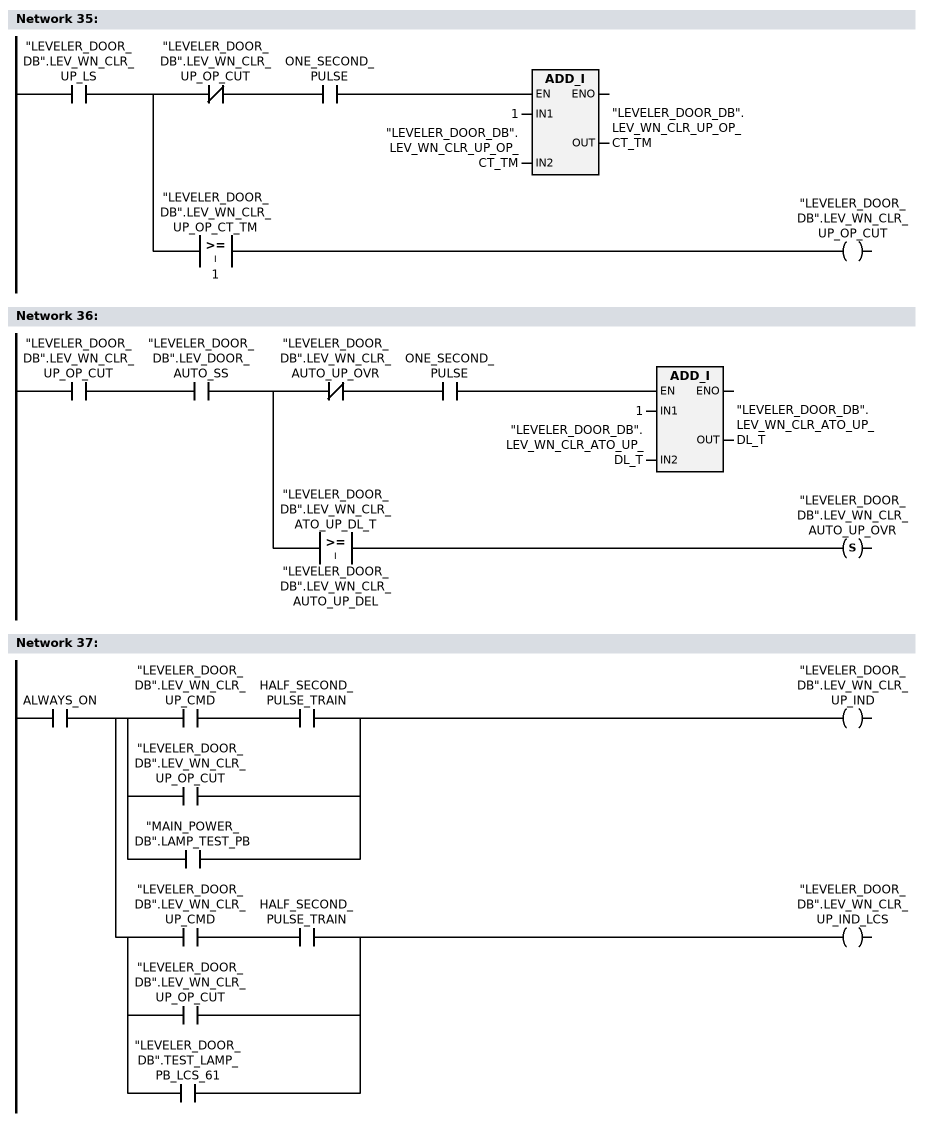
NETWORK
TITLE =
      A     "LEVELER_DOOR_DB".LEV_WN_CLR_UP_LS;
      =     L 0.0;
      A     L 0.0;
      AN    "LEVELER_DOOR_DB".LEV_WN_CLR_UP_OP_CUT;
      A     "ONE_SECOND_PULSE";
      JNB   M033;
      L     1;
      L     "LEVELER_DOOR_DB".LEV_WN_CLR_UP_OP_CT_TM;
      +I;
      T     "LEVELER_DOOR_DB".LEV_WN_CLR_UP_OP_CT_TM;
M033: NOP   0;
      A     L 0.0;
      A(;
      L     "LEVELER_DOOR_DB".LEV_WN_CLR_UP_OP_CT_TM;
      L     1;
      >=I;
      );
      =     "LEVELER_DOOR_DB".LEV_WN_CLR_UP_OP_CUT;
NETWORK
TITLE =
      A     "LEVELER_DOOR_DB".LEV_WN_CLR_UP_OP_CUT;
      A     "LEVELER_DOOR_DB".LEV_DOOR_AUTO_SS;
      =     L 0.0;
      A     L 0.0;
      AN    "LEVELER_DOOR_DB".LEV_WN_CLR_AUTO_UP_OVR;
      A     "ONE_SECOND_PULSE";
      JNB   M034;
      L     1;
      L     "LEVELER_DOOR_DB".LEV_WN_CLR_ATO_UP_DL_T;
      +I;
      T     "LEVELER_DOOR_DB".LEV_WN_CLR_ATO_UP_DL_T;
M034: NOP   0;
      A     L 0.0;
      A(;
      L     "LEVELER_DOOR_DB".LEV_WN_CLR_ATO_UP_DL_T;
      L     "LEVELER_DOOR_DB".LEV_WN_CLR_AUTO_UP_DEL;
      >=I;
      );
      S     "LEVELER_DOOR_DB".LEV_WN_CLR_AUTO_UP_OVR;
NETWORK
TITLE =
      A     "ALWAYS_ON";
      =     L 0.0;
      A     L 0.0;
      A(;
      A     "LEVELER_DOOR_DB".LEV_WN_CLR_UP_CMD;
      A     "HALF_SECOND_PULSE_TRAIN";
      O     "LEVELER_DOOR_DB".LEV_WN_CLR_UP_OP_CUT;
      O     "MAIN_POWER_DB".LAMP_TEST_PB;
      );
      =     "LEVELER_DOOR_DB".LEV_WN_CLR_UP_IND;
      A     L 0.0;
      A(;
      A     "LEVELER_DOOR_DB".LEV_WN_CLR_UP_CMD;
      A     "HALF_SECOND_PULSE_TRAIN";
      O     "LEVELER_DOOR_DB".LEV_WN_CLR_UP_OP_CUT;
      O     "LEVELER_DOOR_DB".TEST_LAMP_PB_LCS_61;
      );
      =     "LEVELER_DOOR_DB".LEV_WN_CLR_UP_IND_LCS;
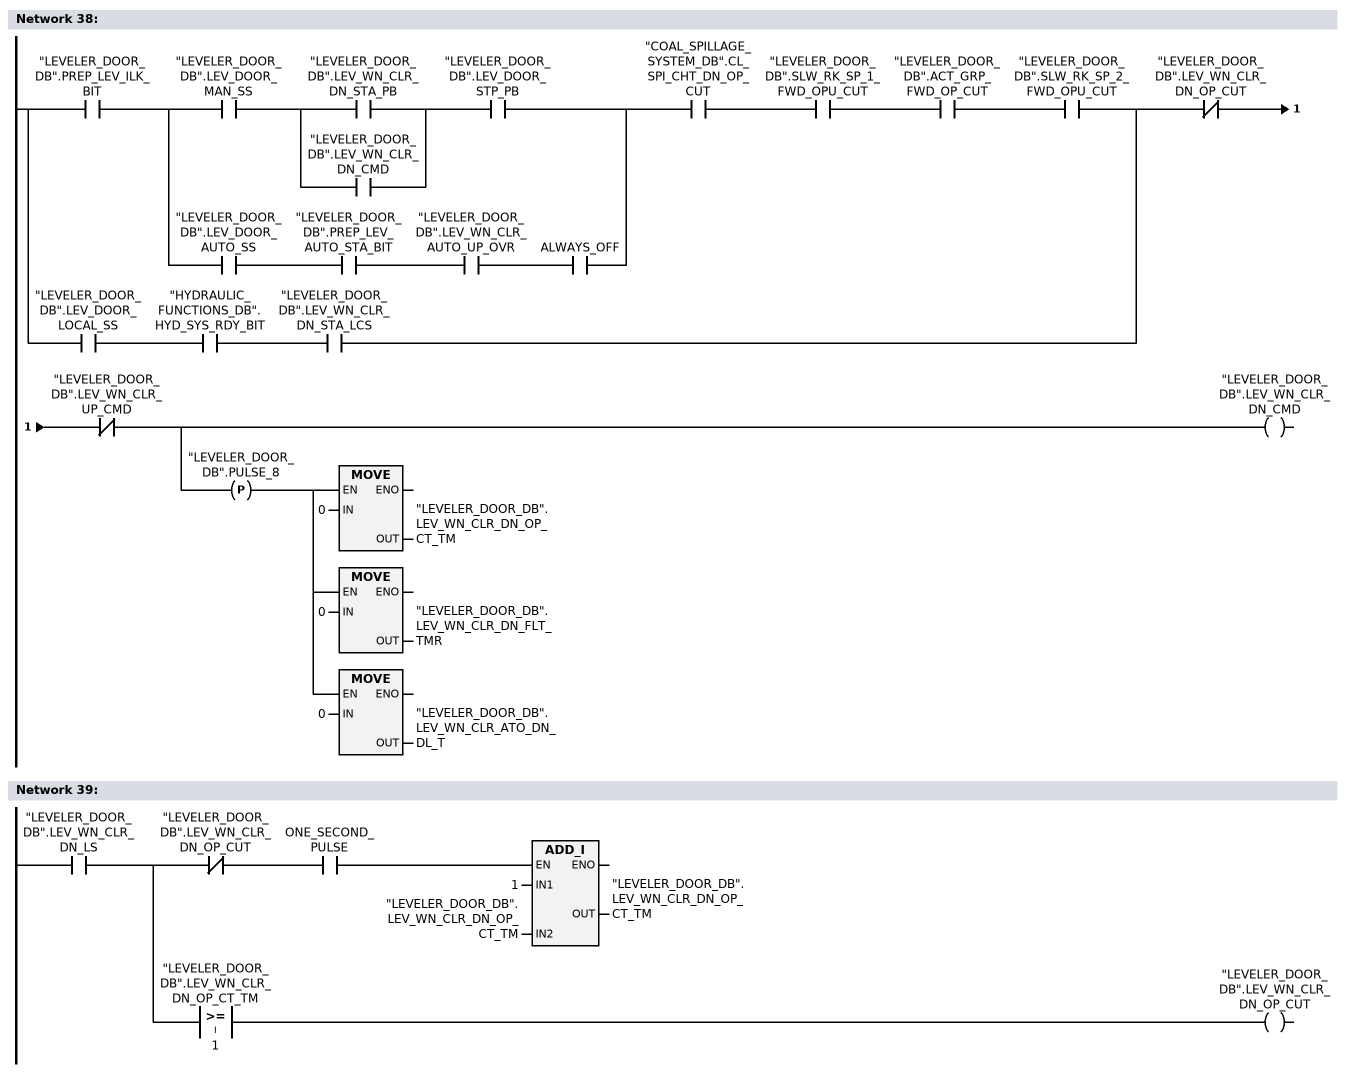
NETWORK
TITLE =
      A(;
      A     "LEVELER_DOOR_DB".PREP_LEV_ILK_BIT;
      A(;
      A     "LEVELER_DOOR_DB".LEV_DOOR_MAN_SS;
      A(;
      O     "LEVELER_DOOR_DB".LEV_WN_CLR_DN_STA_PB;
      O     "LEVELER_DOOR_DB".LEV_WN_CLR_DN_CMD;
      );
      A     "LEVELER_DOOR_DB".LEV_DOOR_STP_PB;
      O;
      A     "LEVELER_DOOR_DB".LEV_DOOR_AUTO_SS;
      A     "LEVELER_DOOR_DB".PREP_LEV_AUTO_STA_BIT;
      A     "LEVELER_DOOR_DB".LEV_WN_CLR_AUTO_UP_OVR;
      A     "ALWAYS_OFF";
      );
      A     "COAL_SPILLAGE_SYSTEM_DB".CL_SPI_CHT_DN_OP_CUT;
      A     "LEVELER_DOOR_DB".SLW_RK_SP_1_FWD_OPU_CUT;
      A     "LEVELER_DOOR_DB".ACT_GRP_FWD_OP_CUT;
      A     "LEVELER_DOOR_DB".SLW_RK_SP_2_FWD_OPU_CUT;
      O;
      A     "LEVELER_DOOR_DB".LEV_DOOR_LOCAL_SS;
      A     "HYDRAULIC_FUNCTIONS_DB".HYD_SYS_RDY_BIT;
      A     "LEVELER_DOOR_DB".LEV_WN_CLR_DN_STA_LCS;
      );
      AN    "LEVELER_DOOR_DB".LEV_WN_CLR_DN_OP_CUT;
      AN    "LEVELER_DOOR_DB".LEV_WN_CLR_UP_CMD;
      =     L 0.0;
      A     L 0.0;
      BLD   102;
      =     "LEVELER_DOOR_DB".LEV_WN_CLR_DN_CMD;
      A     L 0.0;
      FP    "LEVELER_DOOR_DB".PULSE_8;
      =     L 0.1;
      A     L 0.1;
      JNB   M035;
      L     0;
      T     "LEVELER_DOOR_DB".LEV_WN_CLR_DN_OP_CT_TM;
M035: NOP   0;
      A     L 0.1;
      JNB   M036;
      L     0;
      T     "LEVELER_DOOR_DB".LEV_WN_CLR_DN_FLT_TMR;
M036: NOP   0;
      A     L 0.1;
      JNB   M037;
      L     0;
      T     "LEVELER_DOOR_DB".LEV_WN_CLR_ATO_DN_DL_T;
M037: NOP   0;
NETWORK
TITLE =
      A     "LEVELER_DOOR_DB".LEV_WN_CLR_DN_LS;
      =     L 0.0;
      A     L 0.0;
      AN    "LEVELER_DOOR_DB".LEV_WN_CLR_DN_OP_CUT;
      A     "ONE_SECOND_PULSE";
      JNB   M038;
      L     1;
      L     "LEVELER_DOOR_DB".LEV_WN_CLR_DN_OP_CT_TM;
      +I;
      T     "LEVELER_DOOR_DB".LEV_WN_CLR_DN_OP_CT_TM;
M038: NOP   0;
      A     L 0.0;
      A(;
      L     "LEVELER_DOOR_DB".LEV_WN_CLR_DN_OP_CT_TM;
      L     1;
      >=I;
      );
      =     "LEVELER_DOOR_DB".LEV_WN_CLR_DN_OP_CUT;
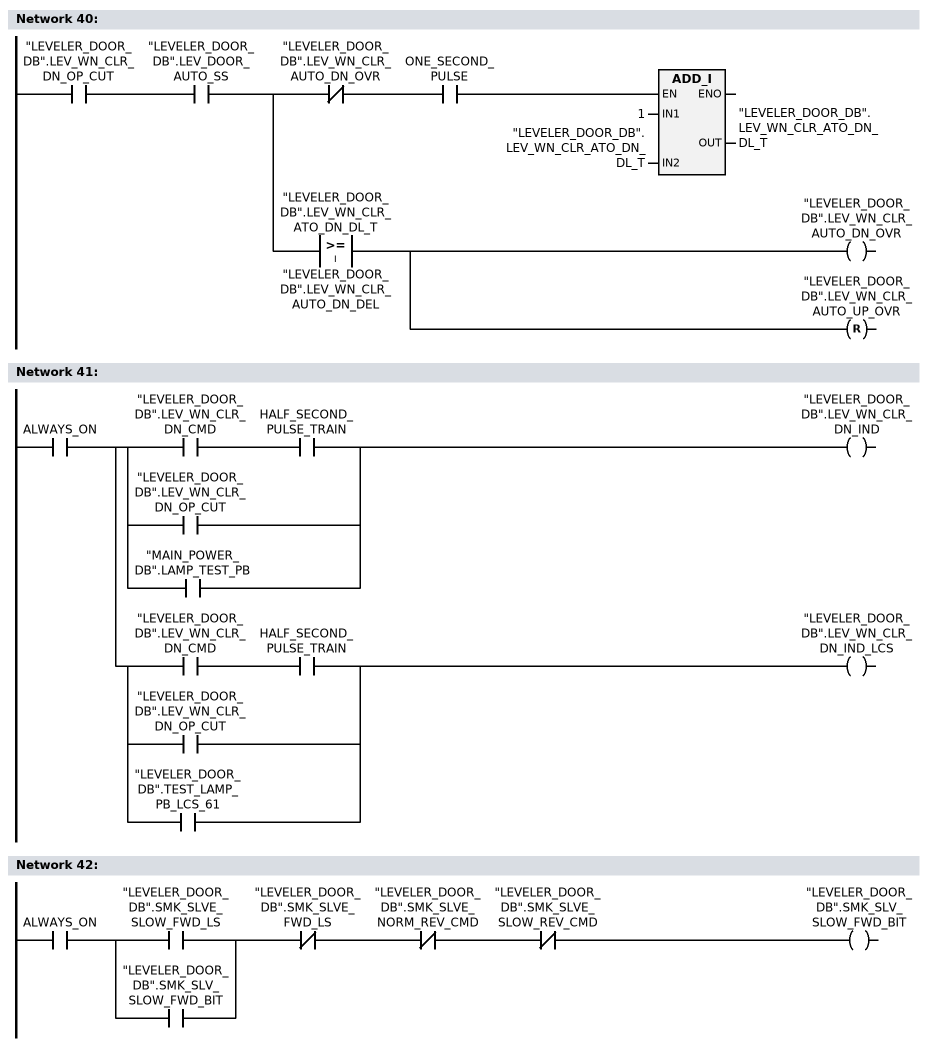
NETWORK
TITLE =
      A     "LEVELER_DOOR_DB".LEV_WN_CLR_DN_OP_CUT;
      A     "LEVELER_DOOR_DB".LEV_DOOR_AUTO_SS;
      =     L 0.0;
      A     L 0.0;
      AN    "LEVELER_DOOR_DB".LEV_WN_CLR_AUTO_DN_OVR;
      A     "ONE_SECOND_PULSE";
      JNB   M039;
      L     1;
      L     "LEVELER_DOOR_DB".LEV_WN_CLR_ATO_DN_DL_T;
      +I;
      T     "LEVELER_DOOR_DB".LEV_WN_CLR_ATO_DN_DL_T;
M039: NOP   0;
      A     L 0.0;
      A(;
      L     "LEVELER_DOOR_DB".LEV_WN_CLR_ATO_DN_DL_T;
      L     "LEVELER_DOOR_DB".LEV_WN_CLR_AUTO_DN_DEL;
      >=I;
      );
      =     "LEVELER_DOOR_DB".LEV_WN_CLR_AUTO_DN_OVR;
      R     "LEVELER_DOOR_DB".LEV_WN_CLR_AUTO_UP_OVR;
NETWORK
TITLE =
      A     "ALWAYS_ON";
      =     L 0.0;
      A     L 0.0;
      A(;
      A     "LEVELER_DOOR_DB".LEV_WN_CLR_DN_CMD;
      A     "HALF_SECOND_PULSE_TRAIN";
      O     "LEVELER_DOOR_DB".LEV_WN_CLR_DN_OP_CUT;
      O     "MAIN_POWER_DB".LAMP_TEST_PB;
      );
      =     "LEVELER_DOOR_DB".LEV_WN_CLR_DN_IND;
      A     L 0.0;
      A(;
      A     "LEVELER_DOOR_DB".LEV_WN_CLR_DN_CMD;
      A     "HALF_SECOND_PULSE_TRAIN";
      O     "LEVELER_DOOR_DB".LEV_WN_CLR_DN_OP_CUT;
      O     "LEVELER_DOOR_DB".TEST_LAMP_PB_LCS_61;
      );
      =     "LEVELER_DOOR_DB".LEV_WN_CLR_DN_IND_LCS;
NETWORK
TITLE =
      A     "ALWAYS_ON";
      A(;
      O     "LEVELER_DOOR_DB".SMK_SLVE_SLOW_FWD_LS;
      O     "LEVELER_DOOR_DB".SMK_SLV_SLOW_FWD_BIT;
      );
      AN    "LEVELER_DOOR_DB".SMK_SLVE_FWD_LS;
      AN    "LEVELER_DOOR_DB".SMK_SLVE_NORM_REV_CMD;
      AN    "LEVELER_DOOR_DB".SMK_SLVE_SLOW_REV_CMD;
      =     "LEVELER_DOOR_DB".SMK_SLV_SLOW_FWD_BIT;
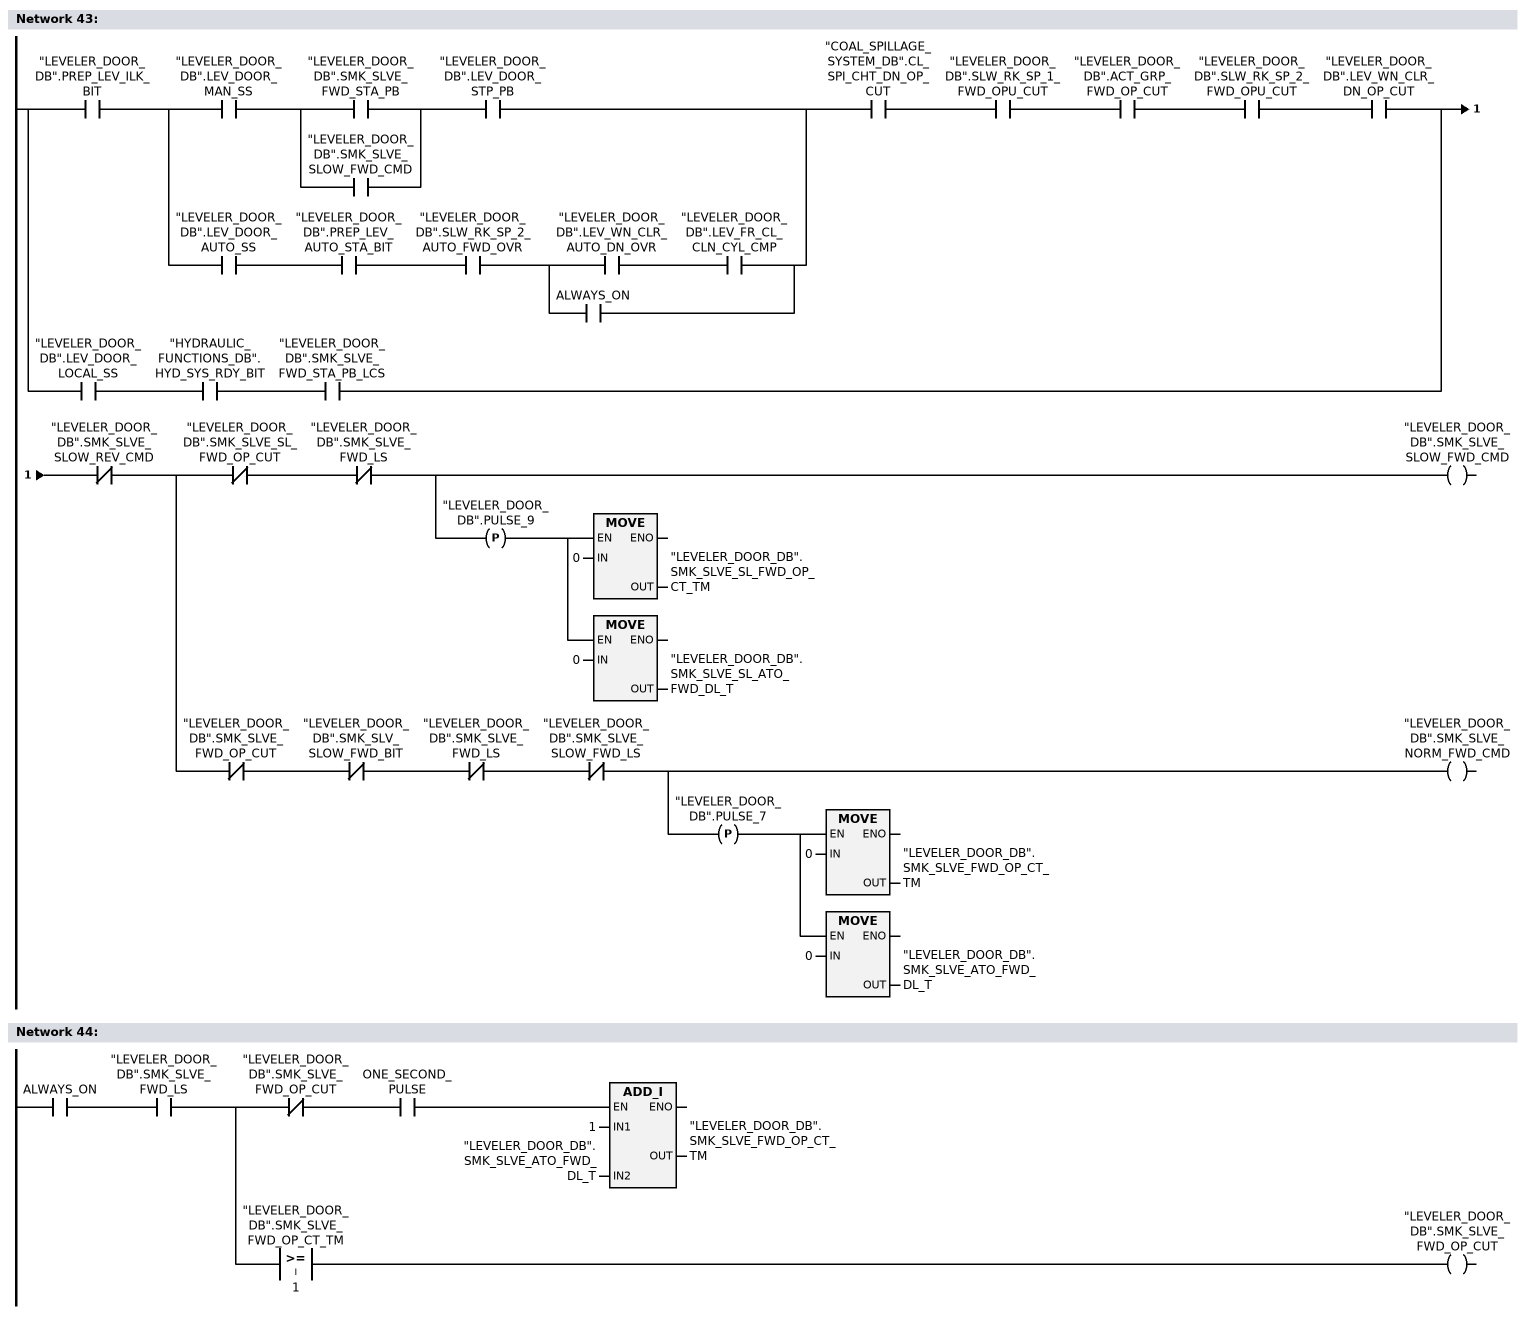
NETWORK
TITLE =
      A(;
      A     "LEVELER_DOOR_DB".PREP_LEV_ILK_BIT;
      A(;
      A     "LEVELER_DOOR_DB".LEV_DOOR_MAN_SS;
      A(;
      O     "LEVELER_DOOR_DB".SMK_SLVE_FWD_STA_PB;
      O     "LEVELER_DOOR_DB".SMK_SLVE_SLOW_FWD_CMD;
      );
      A     "LEVELER_DOOR_DB".LEV_DOOR_STP_PB;
      O;
      A     "LEVELER_DOOR_DB".LEV_DOOR_AUTO_SS;
      A     "LEVELER_DOOR_DB".PREP_LEV_AUTO_STA_BIT;
      A     "LEVELER_DOOR_DB".SLW_RK_SP_2_AUTO_FWD_OVR;
      A(;
      A     "LEVELER_DOOR_DB".LEV_WN_CLR_AUTO_DN_OVR;
      A     "LEVELER_DOOR_DB".LEV_FR_CL_CLN_CYL_CMP;
      O     "ALWAYS_ON";
      );
      );
      A     "COAL_SPILLAGE_SYSTEM_DB".CL_SPI_CHT_DN_OP_CUT;
      A     "LEVELER_DOOR_DB".SLW_RK_SP_1_FWD_OPU_CUT;
      A     "LEVELER_DOOR_DB".ACT_GRP_FWD_OP_CUT;
      A     "LEVELER_DOOR_DB".SLW_RK_SP_2_FWD_OPU_CUT;
      A     "LEVELER_DOOR_DB".LEV_WN_CLR_DN_OP_CUT;
      O;
      A     "LEVELER_DOOR_DB".LEV_DOOR_LOCAL_SS;
      A     "HYDRAULIC_FUNCTIONS_DB".HYD_SYS_RDY_BIT;
      A     "LEVELER_DOOR_DB".SMK_SLVE_FWD_STA_PB_LCS;
      );
      AN    "LEVELER_DOOR_DB".SMK_SLVE_SLOW_REV_CMD;
      =     L 0.0;
      A     L 0.0;
      AN    "LEVELER_DOOR_DB".SMK_SLVE_SL_FWD_OP_CUT;
      AN    "LEVELER_DOOR_DB".SMK_SLVE_FWD_LS;
      =     L 0.1;
      A     L 0.1;
      BLD   102;
      =     "LEVELER_DOOR_DB".SMK_SLVE_SLOW_FWD_CMD;
      A     L 0.1;
      FP    "LEVELER_DOOR_DB".PULSE_9;
      =     L 0.2;
      A     L 0.2;
      JNB   M040;
      L     0;
      T     "LEVELER_DOOR_DB".SMK_SLVE_SL_FWD_OP_CT_TM;
M040: NOP   0;
      A     L 0.2;
      JNB   M041;
      L     0;
      T     "LEVELER_DOOR_DB".SMK_SLVE_SL_ATO_FWD_DL_T;
M041: NOP   0;
      A     L 0.0;
      AN    "LEVELER_DOOR_DB".SMK_SLVE_FWD_OP_CUT;
      AN    "LEVELER_DOOR_DB".SMK_SLV_SLOW_FWD_BIT;
      AN    "LEVELER_DOOR_DB".SMK_SLVE_FWD_LS;
      AN    "LEVELER_DOOR_DB".SMK_SLVE_SLOW_FWD_LS;
      =     L 0.1;
      A     L 0.1;
      BLD   102;
      =     "LEVELER_DOOR_DB".SMK_SLVE_NORM_FWD_CMD;
      A     L 0.1;
      FP    "LEVELER_DOOR_DB".PULSE_7;
      =     L 0.2;
      A     L 0.2;
      JNB   M042;
      L     0;
      T     "LEVELER_DOOR_DB".SMK_SLVE_FWD_OP_CT_TM;
M042: NOP   0;
      A     L 0.2;
      JNB   M043;
      L     0;
      T     "LEVELER_DOOR_DB".SMK_SLVE_ATO_FWD_DL_T;
M043: NOP   0;
NETWORK
TITLE =
      A     "ALWAYS_ON";
      A     "LEVELER_DOOR_DB".SMK_SLVE_FWD_LS;
      =     L 0.0;
      A     L 0.0;
      AN    "LEVELER_DOOR_DB".SMK_SLVE_FWD_OP_CUT;
      A     "ONE_SECOND_PULSE";
      JNB   M044;
      L     1;
      L     "LEVELER_DOOR_DB".SMK_SLVE_ATO_FWD_DL_T;
      +I;
      T     "LEVELER_DOOR_DB".SMK_SLVE_FWD_OP_CT_TM;
M044: NOP   0;
      A     L 0.0;
      A(;
      L     "LEVELER_DOOR_DB".SMK_SLVE_FWD_OP_CT_TM;
      L     1;
      >=I;
      );
      =     "LEVELER_DOOR_DB".SMK_SLVE_FWD_OP_CUT;
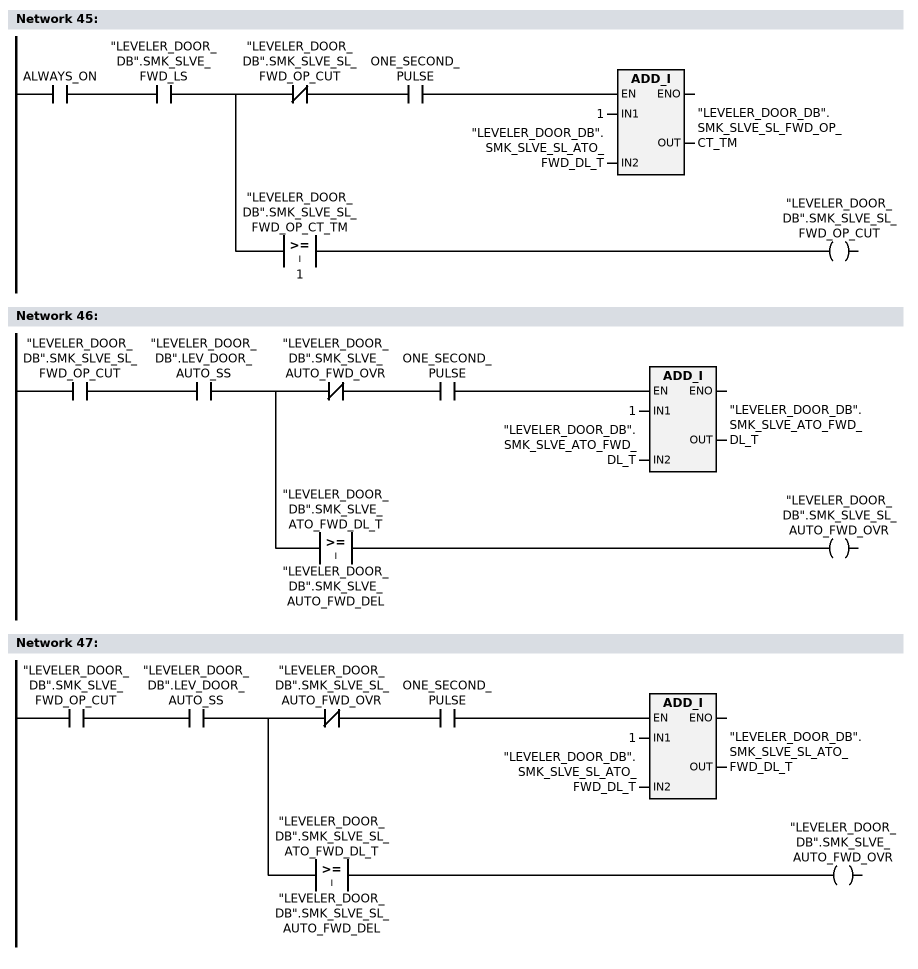
NETWORK
TITLE =
      A     "ALWAYS_ON";
      A     "LEVELER_DOOR_DB".SMK_SLVE_FWD_LS;
      =     L 0.0;
      A     L 0.0;
      AN    "LEVELER_DOOR_DB".SMK_SLVE_SL_FWD_OP_CUT;
      A     "ONE_SECOND_PULSE";
      JNB   M045;
      L     1;
      L     "LEVELER_DOOR_DB".SMK_SLVE_SL_ATO_FWD_DL_T;
      +I;
      T     "LEVELER_DOOR_DB".SMK_SLVE_SL_FWD_OP_CT_TM;
M045: NOP   0;
      A     L 0.0;
      A(;
      L     "LEVELER_DOOR_DB".SMK_SLVE_SL_FWD_OP_CT_TM;
      L     1;
      >=I;
      );
      =     "LEVELER_DOOR_DB".SMK_SLVE_SL_FWD_OP_CUT;
NETWORK
TITLE =
      A     "LEVELER_DOOR_DB".SMK_SLVE_SL_FWD_OP_CUT;
      A     "LEVELER_DOOR_DB".LEV_DOOR_AUTO_SS;
      =     L 0.0;
      A     L 0.0;
      AN    "LEVELER_DOOR_DB".SMK_SLVE_AUTO_FWD_OVR;
      A     "ONE_SECOND_PULSE";
      JNB   M046;
      L     1;
      L     "LEVELER_DOOR_DB".SMK_SLVE_ATO_FWD_DL_T;
      +I;
      T     "LEVELER_DOOR_DB".SMK_SLVE_ATO_FWD_DL_T;
M046: NOP   0;
      A     L 0.0;
      A(;
      L     "LEVELER_DOOR_DB".SMK_SLVE_ATO_FWD_DL_T;
      L     "LEVELER_DOOR_DB".SMK_SLVE_AUTO_FWD_DEL;
      >=I;
      );
      =     "LEVELER_DOOR_DB".SMK_SLVE_SL_AUTO_FWD_OVR;
NETWORK
TITLE =
      A     "LEVELER_DOOR_DB".SMK_SLVE_FWD_OP_CUT;
      A     "LEVELER_DOOR_DB".LEV_DOOR_AUTO_SS;
      =     L 0.0;
      A     L 0.0;
      AN    "LEVELER_DOOR_DB".SMK_SLVE_SL_AUTO_FWD_OVR;
      A     "ONE_SECOND_PULSE";
      JNB   M047;
      L     1;
      L     "LEVELER_DOOR_DB".SMK_SLVE_SL_ATO_FWD_DL_T;
      +I;
      T     "LEVELER_DOOR_DB".SMK_SLVE_SL_ATO_FWD_DL_T;
M047: NOP   0;
      A     L 0.0;
      A(;
      L     "LEVELER_DOOR_DB".SMK_SLVE_SL_ATO_FWD_DL_T;
      L     "LEVELER_DOOR_DB".SMK_SLVE_SL_AUTO_FWD_DEL;
      >=I;
      );
      =     "LEVELER_DOOR_DB".SMK_SLVE_AUTO_FWD_OVR;
